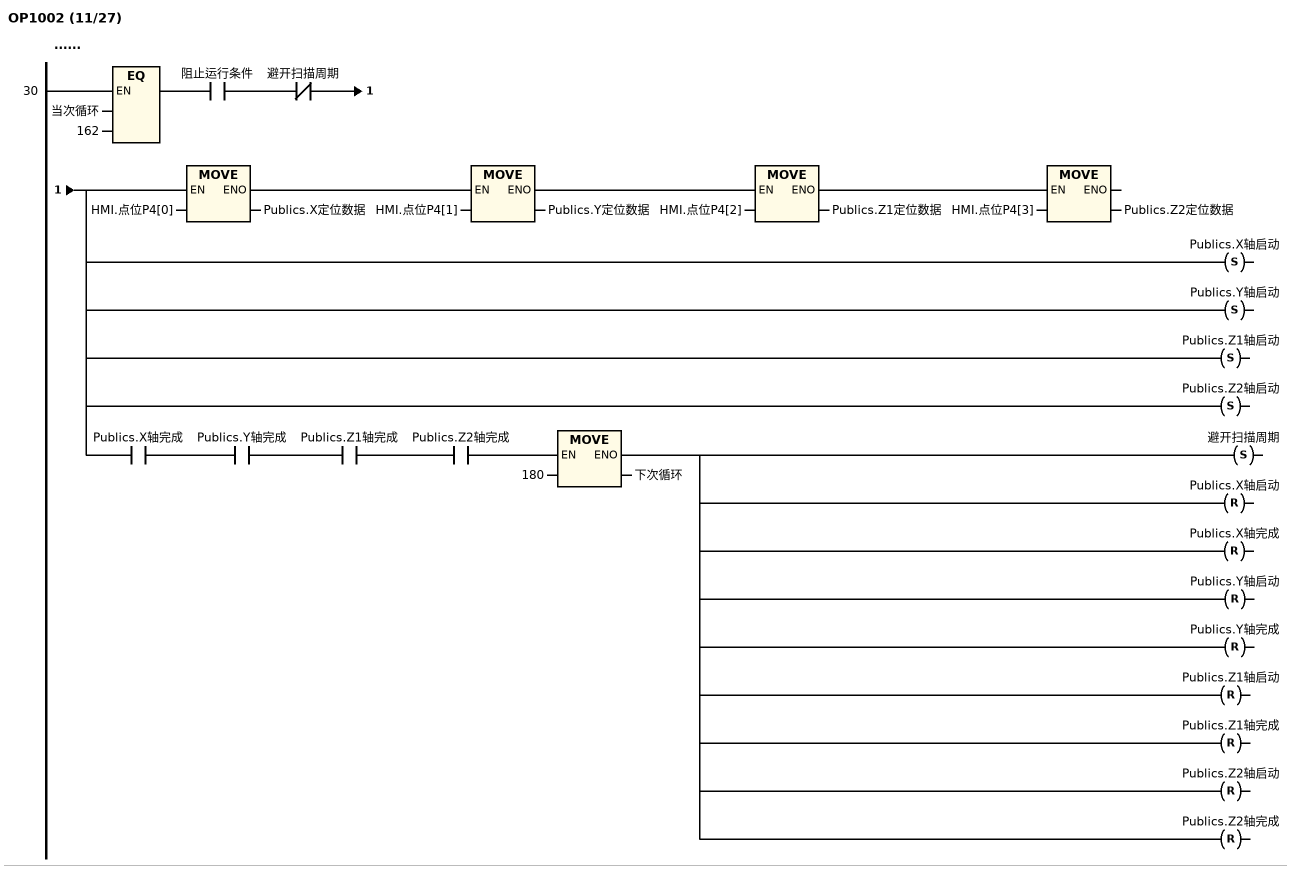
// NETWORK 30: ......
_w32 := 当次循环 = 162 AND 阻止运行条件 AND NOT 避开扫描周期;
IF _w32 THEN Publics.X定位数据 := HMI.点位P4[0]; END_IF
IF _w32 THEN Publics.Y定位数据 := HMI.点位P4[1]; END_IF
IF _w32 THEN Publics.Z1定位数据 := HMI.点位P4[2]; END_IF
IF _w32 THEN Publics.Z2定位数据 := HMI.点位P4[3]; END_IF
Publics.X轴启动 S= _w32;
Publics.Y轴启动 S= _w32;
Publics.Z1轴启动 S= _w32;
Publics.Z2轴启动 S= _w32;
IF _w32 AND Publics.X轴完成 AND Publics.Y轴完成 AND Publics.Z1轴完成 AND Publics.Z2轴完成 THEN 下次循环 := 180; END_IF
_w33 := _w32 AND Publics.X轴完成 AND Publics.Y轴完成 AND Publics.Z1轴完成 AND Publics.Z2轴完成;
避开扫描周期 S= _w33;
Publics.X轴启动 R= _w33;
Publics.X轴完成 R= _w33;
Publics.Y轴启动 R= _w33;
Publics.Y轴完成 R= _w33;
Publics.Z1轴启动 R= _w33;
Publics.Z1轴完成 R= _w33;
Publics.Z2轴启动 R= _w33;
Publics.Z2轴完成 R= _w33;

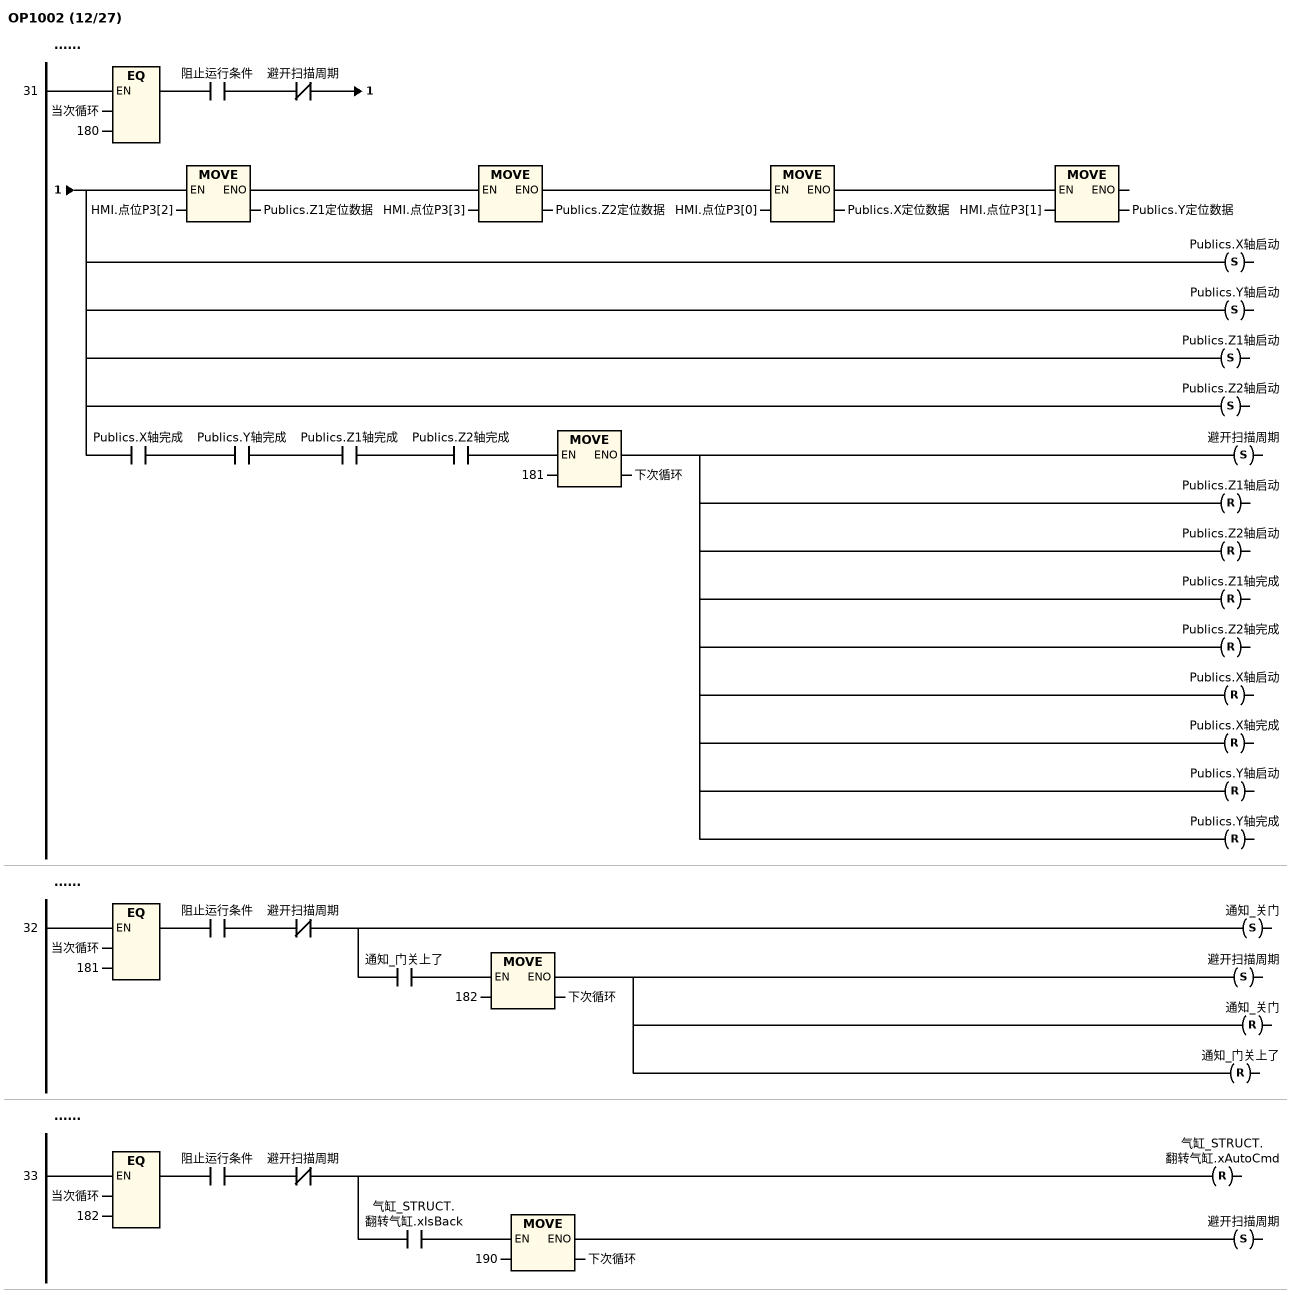
// NETWORK 31: ......
_w34 := 当次循环 = 180 AND 阻止运行条件 AND NOT 避开扫描周期;
IF _w34 THEN Publics.Z1定位数据 := HMI.点位P3[2]; END_IF
IF _w34 THEN Publics.Z2定位数据 := HMI.点位P3[3]; END_IF
IF _w34 THEN Publics.X定位数据 := HMI.点位P3[0]; END_IF
IF _w34 THEN Publics.Y定位数据 := HMI.点位P3[1]; END_IF
Publics.X轴启动 S= _w34;
Publics.Y轴启动 S= _w34;
Publics.Z1轴启动 S= _w34;
Publics.Z2轴启动 S= _w34;
IF _w34 AND Publics.X轴完成 AND Publics.Y轴完成 AND Publics.Z1轴完成 AND Publics.Z2轴完成 THEN 下次循环 := 181; END_IF
_w35 := _w34 AND Publics.X轴完成 AND Publics.Y轴完成 AND Publics.Z1轴完成 AND Publics.Z2轴完成;
避开扫描周期 S= _w35;
Publics.Z1轴启动 R= _w35;
Publics.Z2轴启动 R= _w35;
Publics.Z1轴完成 R= _w35;
Publics.Z2轴完成 R= _w35;
Publics.X轴启动 R= _w35;
Publics.X轴完成 R= _w35;
Publics.Y轴启动 R= _w35;
Publics.Y轴完成 R= _w35;

// NETWORK 32: ......
_w36 := 当次循环 = 181 AND 阻止运行条件 AND NOT 避开扫描周期;
通知_关门 S= _w36;
IF _w36 AND 通知_门关上了 THEN 下次循环 := 182; END_IF
_w37 := _w36 AND 通知_门关上了;
避开扫描周期 S= _w37;
通知_关门 R= _w37;
通知_门关上了 R= _w37;

// NETWORK 33: ......
_w38 := 当次循环 = 182 AND 阻止运行条件 AND NOT 避开扫描周期;
气缸_STRUCT.翻转气缸.xAutoCmd R= _w38;
IF _w38 AND 气缸_STRUCT.翻转气缸.xIsBack THEN 下次循环 := 190; END_IF
避开扫描周期 S= _w38 AND 气缸_STRUCT.翻转气缸.xIsBack;

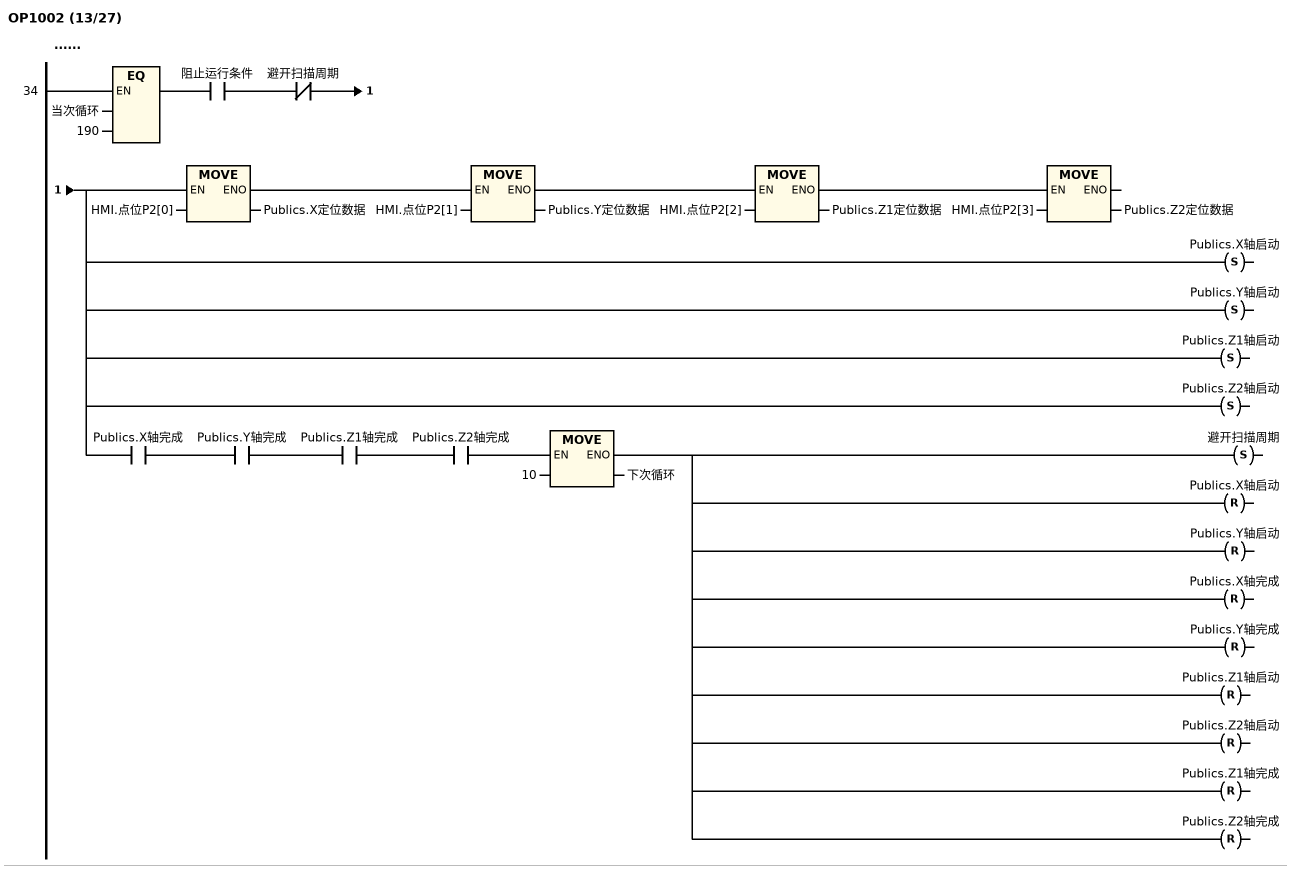
// NETWORK 34: ......
_w39 := 当次循环 = 190 AND 阻止运行条件 AND NOT 避开扫描周期;
IF _w39 THEN Publics.X定位数据 := HMI.点位P2[0]; END_IF
IF _w39 THEN Publics.Y定位数据 := HMI.点位P2[1]; END_IF
IF _w39 THEN Publics.Z1定位数据 := HMI.点位P2[2]; END_IF
IF _w39 THEN Publics.Z2定位数据 := HMI.点位P2[3]; END_IF
Publics.X轴启动 S= _w39;
Publics.Y轴启动 S= _w39;
Publics.Z1轴启动 S= _w39;
Publics.Z2轴启动 S= _w39;
IF _w39 AND Publics.X轴完成 AND Publics.Y轴完成 AND Publics.Z1轴完成 AND Publics.Z2轴完成 THEN 下次循环 := 10; END_IF
_w40 := _w39 AND Publics.X轴完成 AND Publics.Y轴完成 AND Publics.Z1轴完成 AND Publics.Z2轴完成;
避开扫描周期 S= _w40;
Publics.X轴启动 R= _w40;
Publics.Y轴启动 R= _w40;
Publics.X轴完成 R= _w40;
Publics.Y轴完成 R= _w40;
Publics.Z1轴启动 R= _w40;
Publics.Z2轴启动 R= _w40;
Publics.Z1轴完成 R= _w40;
Publics.Z2轴完成 R= _w40;

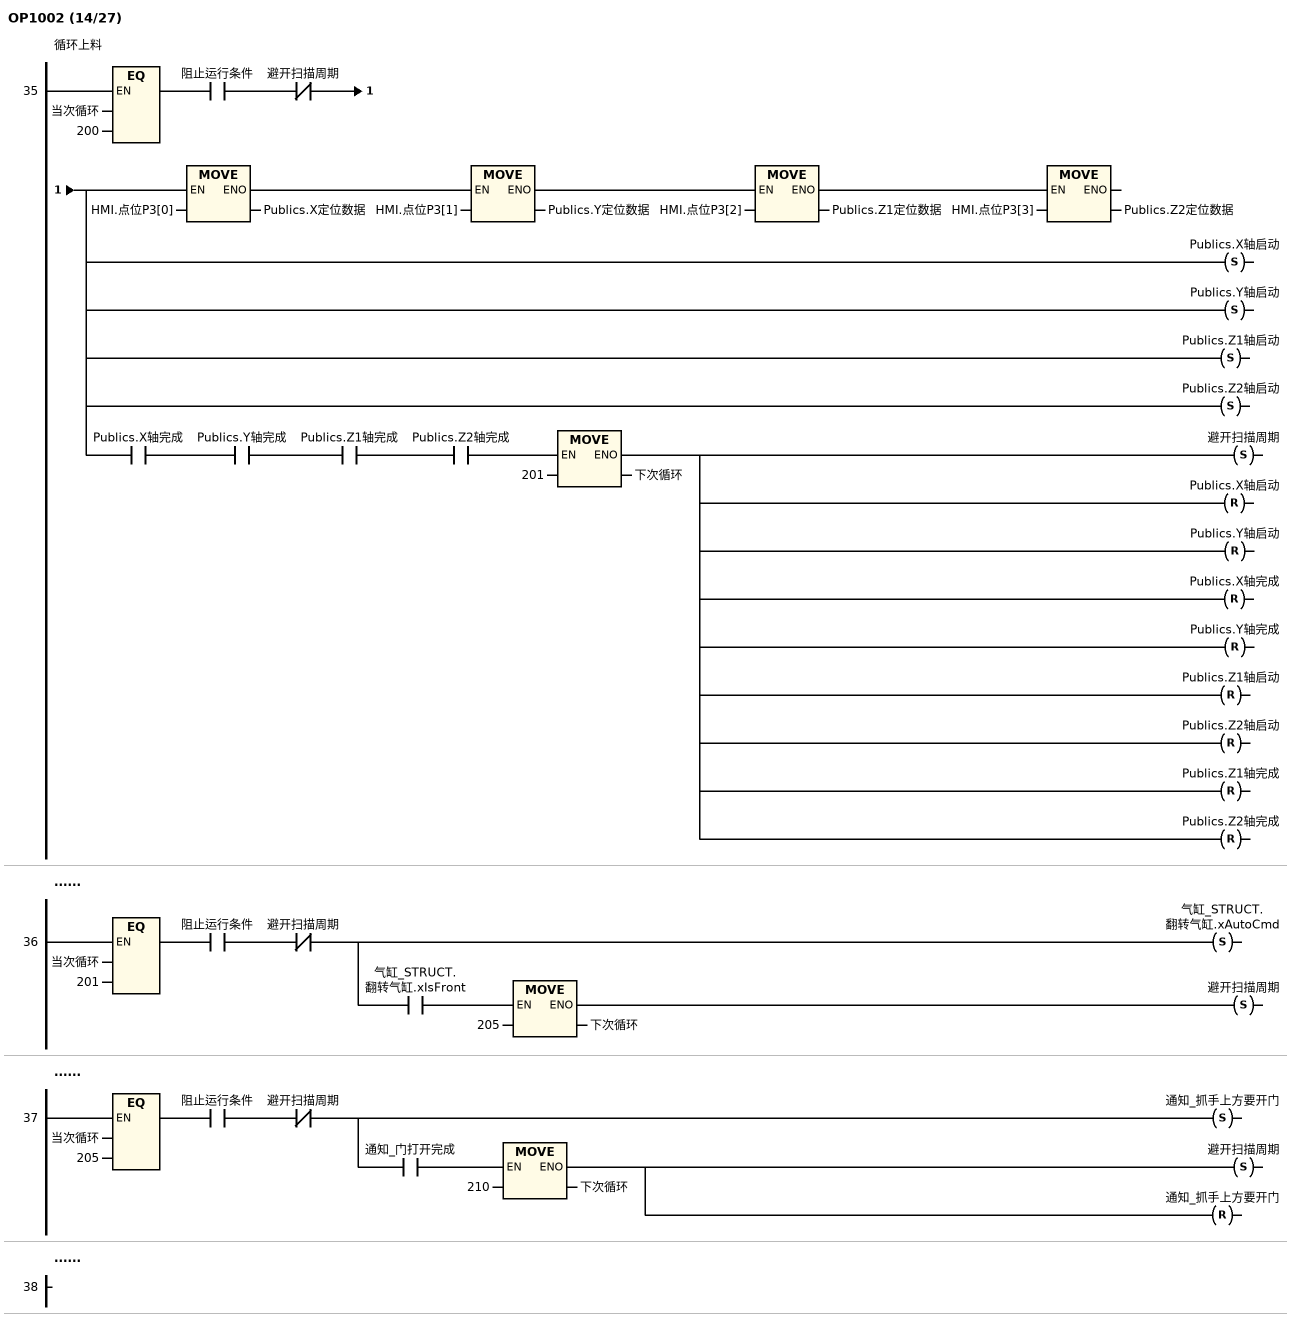
// NETWORK 35: 循环上料
_w41 := 当次循环 = 200 AND 阻止运行条件 AND NOT 避开扫描周期;
IF _w41 THEN Publics.X定位数据 := HMI.点位P3[0]; END_IF
IF _w41 THEN Publics.Y定位数据 := HMI.点位P3[1]; END_IF
IF _w41 THEN Publics.Z1定位数据 := HMI.点位P3[2]; END_IF
IF _w41 THEN Publics.Z2定位数据 := HMI.点位P3[3]; END_IF
Publics.X轴启动 S= _w41;
Publics.Y轴启动 S= _w41;
Publics.Z1轴启动 S= _w41;
Publics.Z2轴启动 S= _w41;
IF _w41 AND Publics.X轴完成 AND Publics.Y轴完成 AND Publics.Z1轴完成 AND Publics.Z2轴完成 THEN 下次循环 := 201; END_IF
_w42 := _w41 AND Publics.X轴完成 AND Publics.Y轴完成 AND Publics.Z1轴完成 AND Publics.Z2轴完成;
避开扫描周期 S= _w42;
Publics.X轴启动 R= _w42;
Publics.Y轴启动 R= _w42;
Publics.X轴完成 R= _w42;
Publics.Y轴完成 R= _w42;
Publics.Z1轴启动 R= _w42;
Publics.Z2轴启动 R= _w42;
Publics.Z1轴完成 R= _w42;
Publics.Z2轴完成 R= _w42;

// NETWORK 36: ......
_w43 := 当次循环 = 201 AND 阻止运行条件 AND NOT 避开扫描周期;
气缸_STRUCT.翻转气缸.xAutoCmd S= _w43;
IF _w43 AND 气缸_STRUCT.翻转气缸.xIsFront THEN 下次循环 := 205; END_IF
避开扫描周期 S= _w43 AND 气缸_STRUCT.翻转气缸.xIsFront;

// NETWORK 37: ......
_w44 := 当次循环 = 205 AND 阻止运行条件 AND NOT 避开扫描周期;
通知_抓手上方要开门 S= _w44;
IF _w44 AND 通知_门打开完成 THEN 下次循环 := 210; END_IF
_w45 := _w44 AND 通知_门打开完成;
避开扫描周期 S= _w45;
通知_抓手上方要开门 R= _w45;

// NETWORK 38: ......

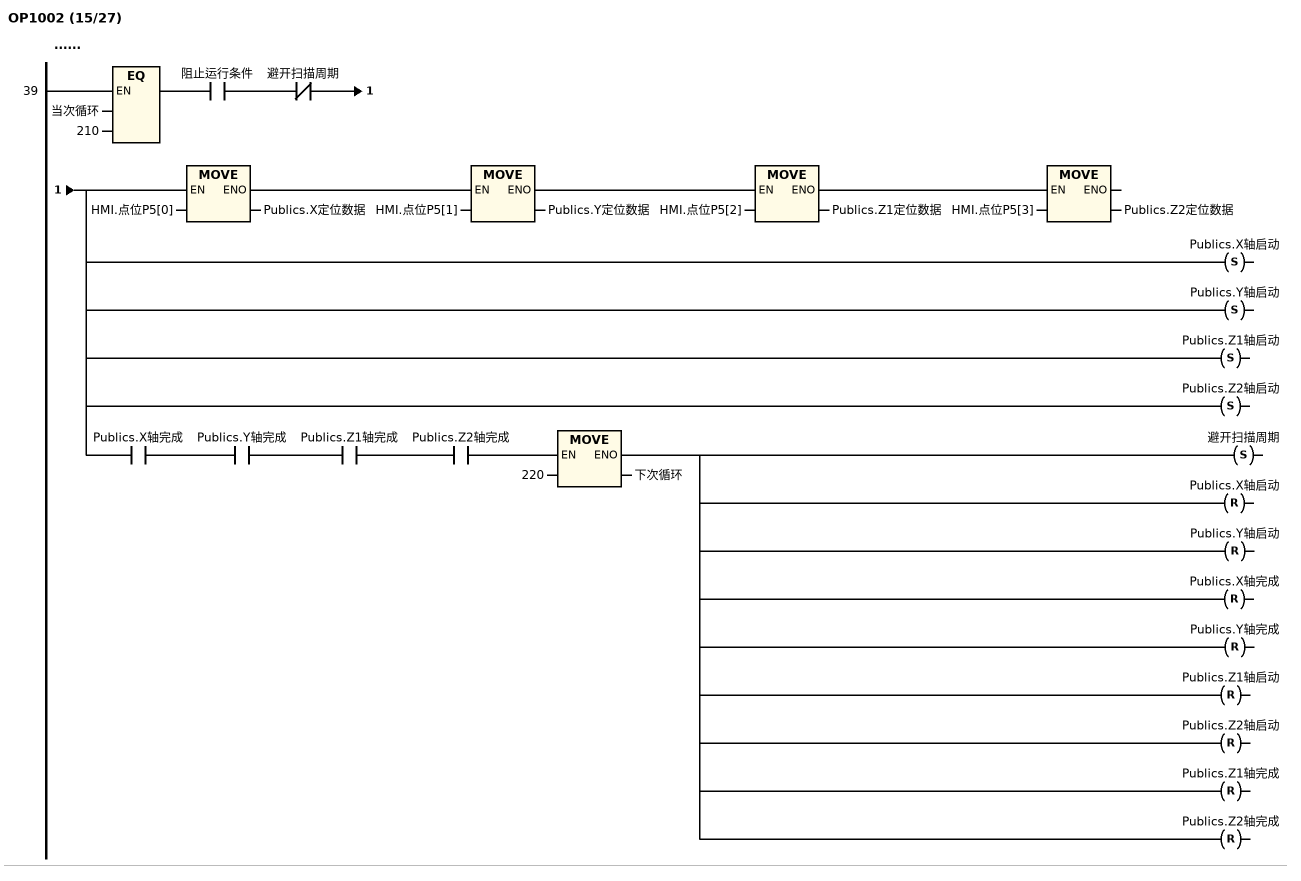
// NETWORK 39: ......
_w46 := 当次循环 = 210 AND 阻止运行条件 AND NOT 避开扫描周期;
IF _w46 THEN Publics.X定位数据 := HMI.点位P5[0]; END_IF
IF _w46 THEN Publics.Y定位数据 := HMI.点位P5[1]; END_IF
IF _w46 THEN Publics.Z1定位数据 := HMI.点位P5[2]; END_IF
IF _w46 THEN Publics.Z2定位数据 := HMI.点位P5[3]; END_IF
Publics.X轴启动 S= _w46;
Publics.Y轴启动 S= _w46;
Publics.Z1轴启动 S= _w46;
Publics.Z2轴启动 S= _w46;
IF _w46 AND Publics.X轴完成 AND Publics.Y轴完成 AND Publics.Z1轴完成 AND Publics.Z2轴完成 THEN 下次循环 := 220; END_IF
_w47 := _w46 AND Publics.X轴完成 AND Publics.Y轴完成 AND Publics.Z1轴完成 AND Publics.Z2轴完成;
避开扫描周期 S= _w47;
Publics.X轴启动 R= _w47;
Publics.Y轴启动 R= _w47;
Publics.X轴完成 R= _w47;
Publics.Y轴完成 R= _w47;
Publics.Z1轴启动 R= _w47;
Publics.Z2轴启动 R= _w47;
Publics.Z1轴完成 R= _w47;
Publics.Z2轴完成 R= _w47;

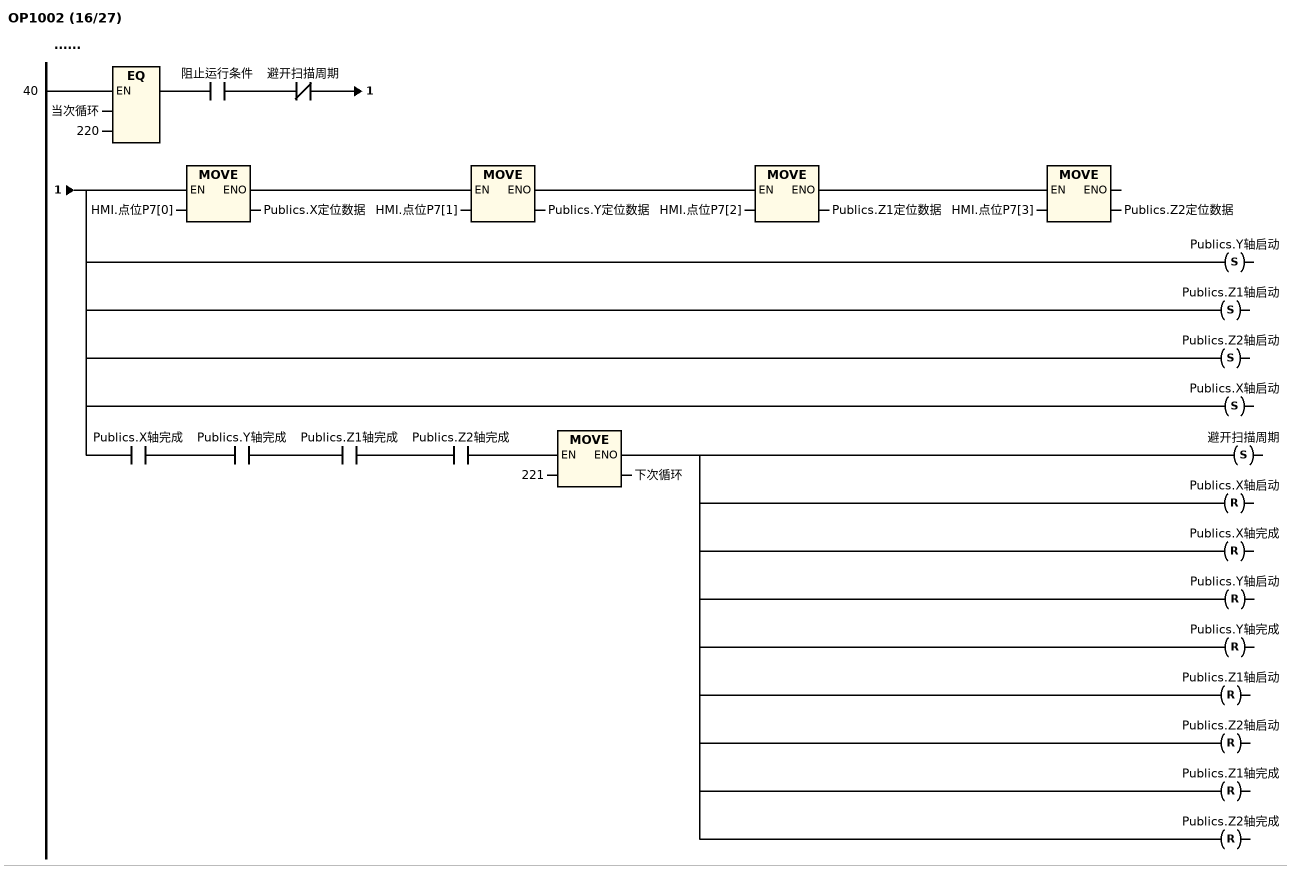
// NETWORK 40: ......
_w48 := 当次循环 = 220 AND 阻止运行条件 AND NOT 避开扫描周期;
IF _w48 THEN Publics.X定位数据 := HMI.点位P7[0]; END_IF
IF _w48 THEN Publics.Y定位数据 := HMI.点位P7[1]; END_IF
IF _w48 THEN Publics.Z1定位数据 := HMI.点位P7[2]; END_IF
IF _w48 THEN Publics.Z2定位数据 := HMI.点位P7[3]; END_IF
Publics.Y轴启动 S= _w48;
Publics.Z1轴启动 S= _w48;
Publics.Z2轴启动 S= _w48;
Publics.X轴启动 S= _w48;
IF _w48 AND Publics.X轴完成 AND Publics.Y轴完成 AND Publics.Z1轴完成 AND Publics.Z2轴完成 THEN 下次循环 := 221; END_IF
_w49 := _w48 AND Publics.X轴完成 AND Publics.Y轴完成 AND Publics.Z1轴完成 AND Publics.Z2轴完成;
避开扫描周期 S= _w49;
Publics.X轴启动 R= _w49;
Publics.X轴完成 R= _w49;
Publics.Y轴启动 R= _w49;
Publics.Y轴完成 R= _w49;
Publics.Z1轴启动 R= _w49;
Publics.Z2轴启动 R= _w49;
Publics.Z1轴完成 R= _w49;
Publics.Z2轴完成 R= _w49;

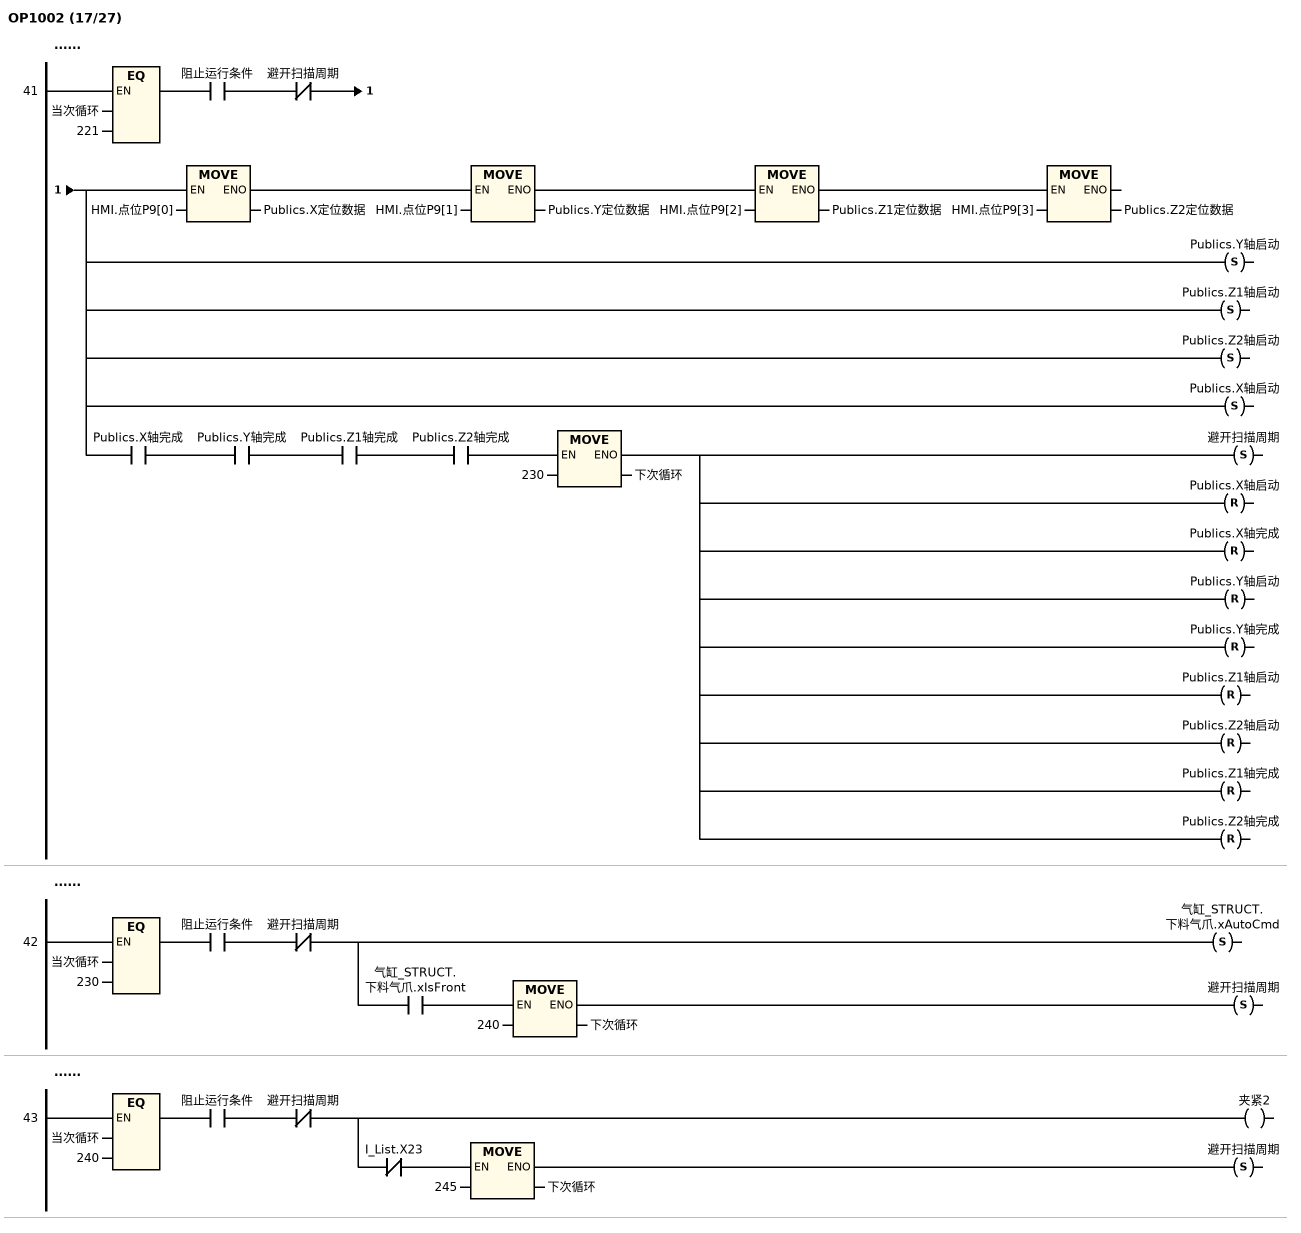
// NETWORK 41: ......
_w50 := 当次循环 = 221 AND 阻止运行条件 AND NOT 避开扫描周期;
IF _w50 THEN Publics.X定位数据 := HMI.点位P9[0]; END_IF
IF _w50 THEN Publics.Y定位数据 := HMI.点位P9[1]; END_IF
IF _w50 THEN Publics.Z1定位数据 := HMI.点位P9[2]; END_IF
IF _w50 THEN Publics.Z2定位数据 := HMI.点位P9[3]; END_IF
Publics.Y轴启动 S= _w50;
Publics.Z1轴启动 S= _w50;
Publics.Z2轴启动 S= _w50;
Publics.X轴启动 S= _w50;
IF _w50 AND Publics.X轴完成 AND Publics.Y轴完成 AND Publics.Z1轴完成 AND Publics.Z2轴完成 THEN 下次循环 := 230; END_IF
_w51 := _w50 AND Publics.X轴完成 AND Publics.Y轴完成 AND Publics.Z1轴完成 AND Publics.Z2轴完成;
避开扫描周期 S= _w51;
Publics.X轴启动 R= _w51;
Publics.X轴完成 R= _w51;
Publics.Y轴启动 R= _w51;
Publics.Y轴完成 R= _w51;
Publics.Z1轴启动 R= _w51;
Publics.Z2轴启动 R= _w51;
Publics.Z1轴完成 R= _w51;
Publics.Z2轴完成 R= _w51;

// NETWORK 42: ......
_w52 := 当次循环 = 230 AND 阻止运行条件 AND NOT 避开扫描周期;
气缸_STRUCT.下料气爪.xAutoCmd S= _w52;
IF _w52 AND 气缸_STRUCT.下料气爪.xIsFront THEN 下次循环 := 240; END_IF
避开扫描周期 S= _w52 AND 气缸_STRUCT.下料气爪.xIsFront;

// NETWORK 43: ......
_w53 := 当次循环 = 240 AND 阻止运行条件 AND NOT 避开扫描周期;
夹紧2 := _w53;
IF _w53 AND NOT I_List.X23 THEN 下次循环 := 245; END_IF
避开扫描周期 S= _w53 AND NOT I_List.X23;

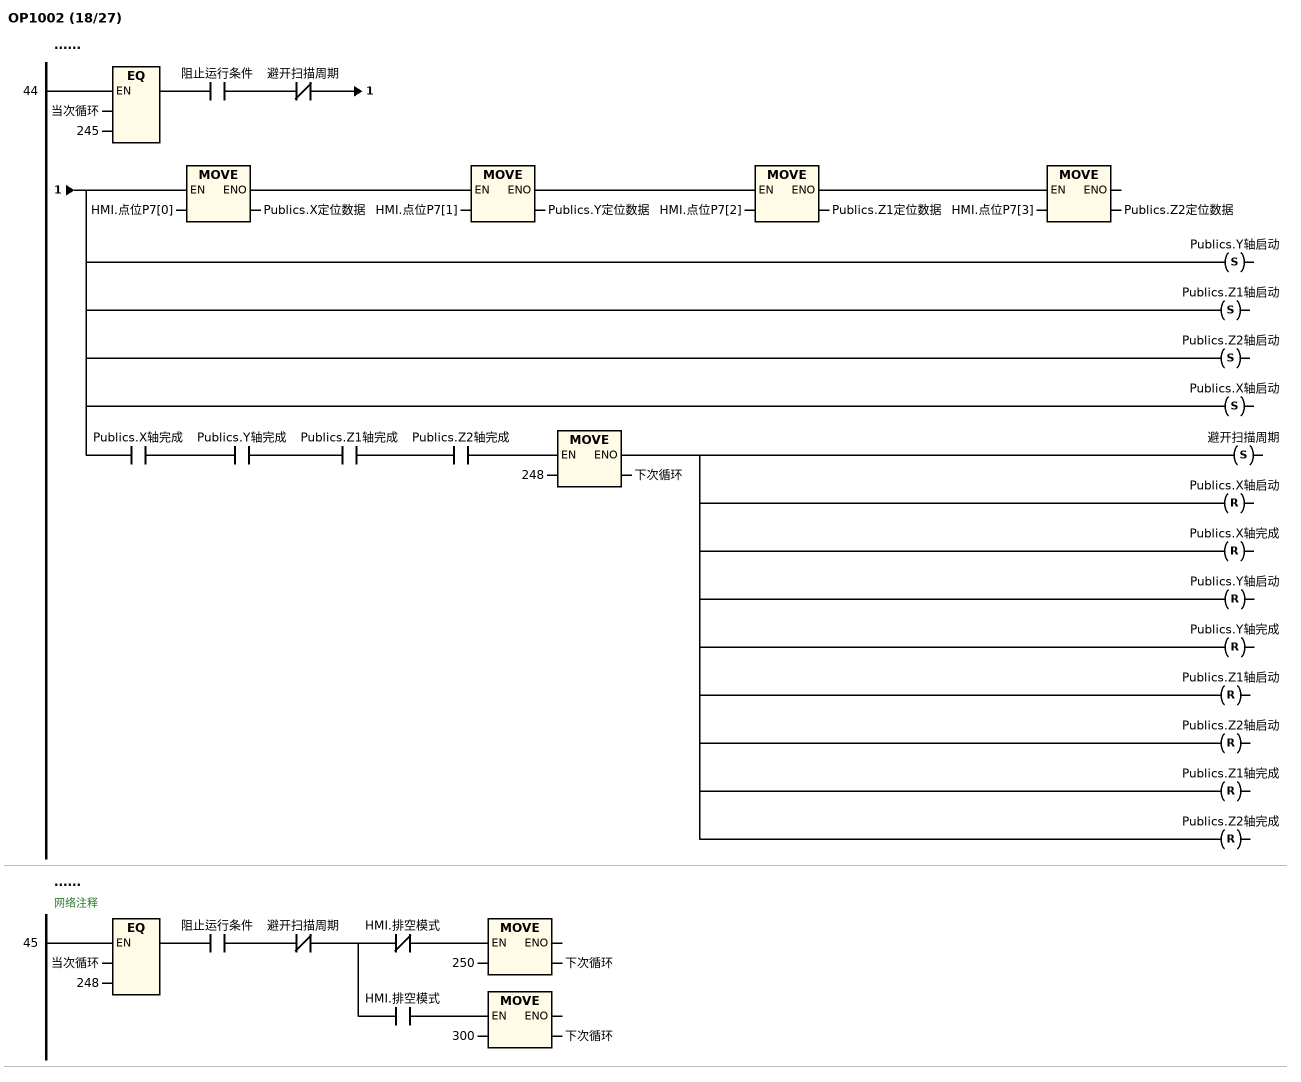
// NETWORK 44: ......
_w54 := 当次循环 = 245 AND 阻止运行条件 AND NOT 避开扫描周期;
IF _w54 THEN Publics.X定位数据 := HMI.点位P7[0]; END_IF
IF _w54 THEN Publics.Y定位数据 := HMI.点位P7[1]; END_IF
IF _w54 THEN Publics.Z1定位数据 := HMI.点位P7[2]; END_IF
IF _w54 THEN Publics.Z2定位数据 := HMI.点位P7[3]; END_IF
Publics.Y轴启动 S= _w54;
Publics.Z1轴启动 S= _w54;
Publics.Z2轴启动 S= _w54;
Publics.X轴启动 S= _w54;
IF _w54 AND Publics.X轴完成 AND Publics.Y轴完成 AND Publics.Z1轴完成 AND Publics.Z2轴完成 THEN 下次循环 := 248; END_IF
_w55 := _w54 AND Publics.X轴完成 AND Publics.Y轴完成 AND Publics.Z1轴完成 AND Publics.Z2轴完成;
避开扫描周期 S= _w55;
Publics.X轴启动 R= _w55;
Publics.X轴完成 R= _w55;
Publics.Y轴启动 R= _w55;
Publics.Y轴完成 R= _w55;
Publics.Z1轴启动 R= _w55;
Publics.Z2轴启动 R= _w55;
Publics.Z1轴完成 R= _w55;
Publics.Z2轴完成 R= _w55;

// NETWORK 45: ......
// 网络注释
_w56 := 当次循环 = 248 AND 阻止运行条件 AND NOT 避开扫描周期;
IF _w56 AND NOT HMI.排空模式 THEN 下次循环 := 250; END_IF
IF _w56 AND HMI.排空模式 THEN 下次循环 := 300; END_IF

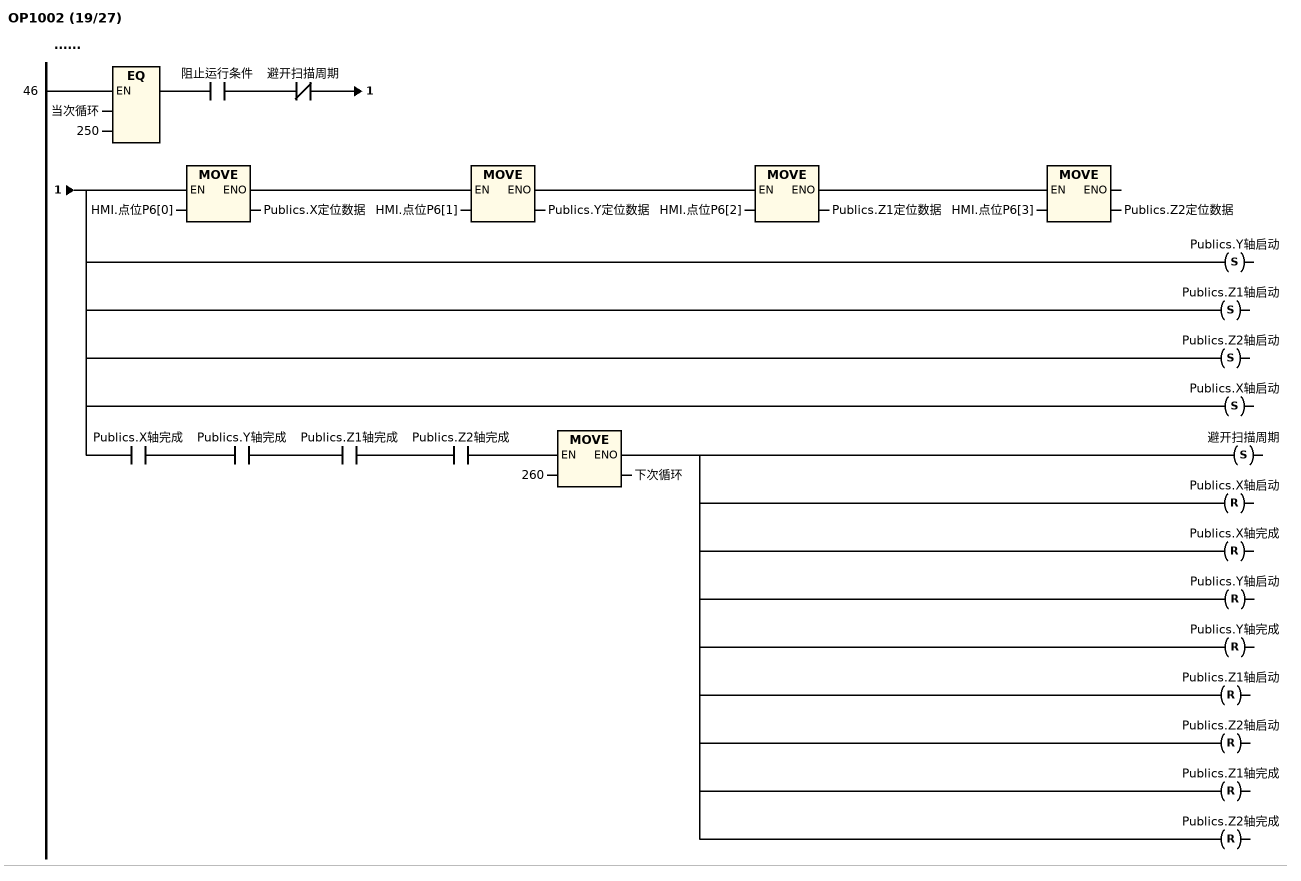
// NETWORK 46: ......
_w57 := 当次循环 = 250 AND 阻止运行条件 AND NOT 避开扫描周期;
IF _w57 THEN Publics.X定位数据 := HMI.点位P6[0]; END_IF
IF _w57 THEN Publics.Y定位数据 := HMI.点位P6[1]; END_IF
IF _w57 THEN Publics.Z1定位数据 := HMI.点位P6[2]; END_IF
IF _w57 THEN Publics.Z2定位数据 := HMI.点位P6[3]; END_IF
Publics.Y轴启动 S= _w57;
Publics.Z1轴启动 S= _w57;
Publics.Z2轴启动 S= _w57;
Publics.X轴启动 S= _w57;
IF _w57 AND Publics.X轴完成 AND Publics.Y轴完成 AND Publics.Z1轴完成 AND Publics.Z2轴完成 THEN 下次循环 := 260; END_IF
_w58 := _w57 AND Publics.X轴完成 AND Publics.Y轴完成 AND Publics.Z1轴完成 AND Publics.Z2轴完成;
避开扫描周期 S= _w58;
Publics.X轴启动 R= _w58;
Publics.X轴完成 R= _w58;
Publics.Y轴启动 R= _w58;
Publics.Y轴完成 R= _w58;
Publics.Z1轴启动 R= _w58;
Publics.Z2轴启动 R= _w58;
Publics.Z1轴完成 R= _w58;
Publics.Z2轴完成 R= _w58;

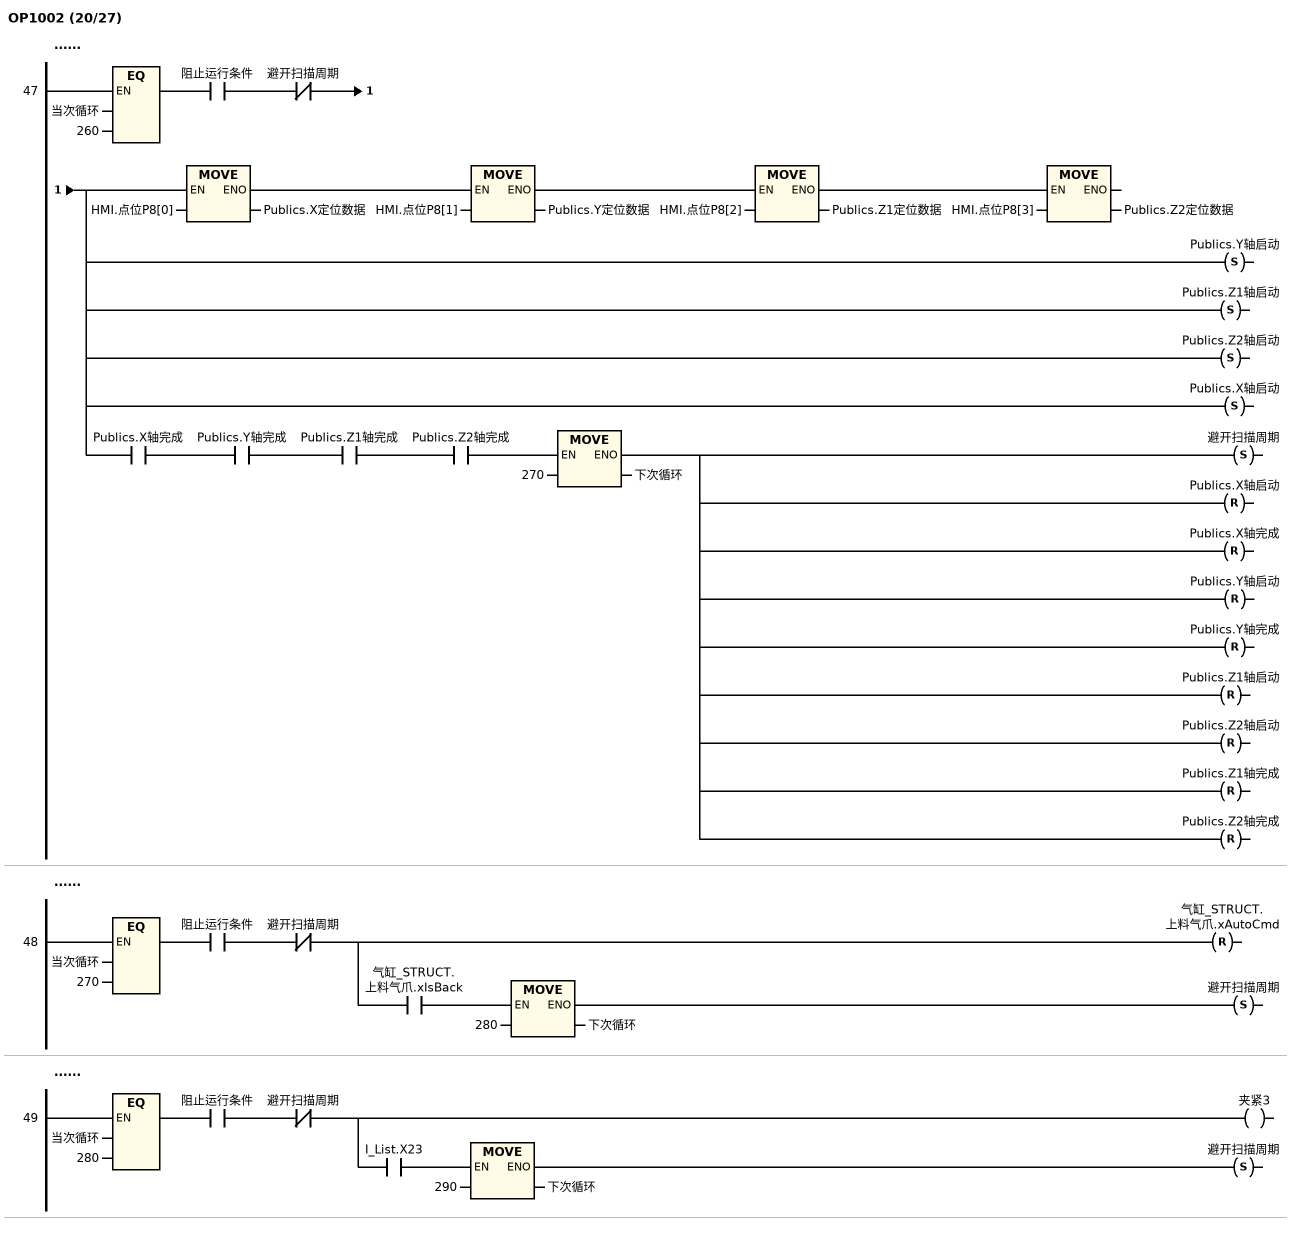
// NETWORK 47: ......
_w59 := 当次循环 = 260 AND 阻止运行条件 AND NOT 避开扫描周期;
IF _w59 THEN Publics.X定位数据 := HMI.点位P8[0]; END_IF
IF _w59 THEN Publics.Y定位数据 := HMI.点位P8[1]; END_IF
IF _w59 THEN Publics.Z1定位数据 := HMI.点位P8[2]; END_IF
IF _w59 THEN Publics.Z2定位数据 := HMI.点位P8[3]; END_IF
Publics.Y轴启动 S= _w59;
Publics.Z1轴启动 S= _w59;
Publics.Z2轴启动 S= _w59;
Publics.X轴启动 S= _w59;
IF _w59 AND Publics.X轴完成 AND Publics.Y轴完成 AND Publics.Z1轴完成 AND Publics.Z2轴完成 THEN 下次循环 := 270; END_IF
_w60 := _w59 AND Publics.X轴完成 AND Publics.Y轴完成 AND Publics.Z1轴完成 AND Publics.Z2轴完成;
避开扫描周期 S= _w60;
Publics.X轴启动 R= _w60;
Publics.X轴完成 R= _w60;
Publics.Y轴启动 R= _w60;
Publics.Y轴完成 R= _w60;
Publics.Z1轴启动 R= _w60;
Publics.Z2轴启动 R= _w60;
Publics.Z1轴完成 R= _w60;
Publics.Z2轴完成 R= _w60;

// NETWORK 48: ......
_w61 := 当次循环 = 270 AND 阻止运行条件 AND NOT 避开扫描周期;
气缸_STRUCT.上料气爪.xAutoCmd R= _w61;
IF _w61 AND 气缸_STRUCT.上料气爪.xIsBack THEN 下次循环 := 280; END_IF
避开扫描周期 S= _w61 AND 气缸_STRUCT.上料气爪.xIsBack;

// NETWORK 49: ......
_w62 := 当次循环 = 280 AND 阻止运行条件 AND NOT 避开扫描周期;
夹紧3 := _w62;
IF _w62 AND I_List.X23 THEN 下次循环 := 290; END_IF
避开扫描周期 S= _w62 AND I_List.X23;

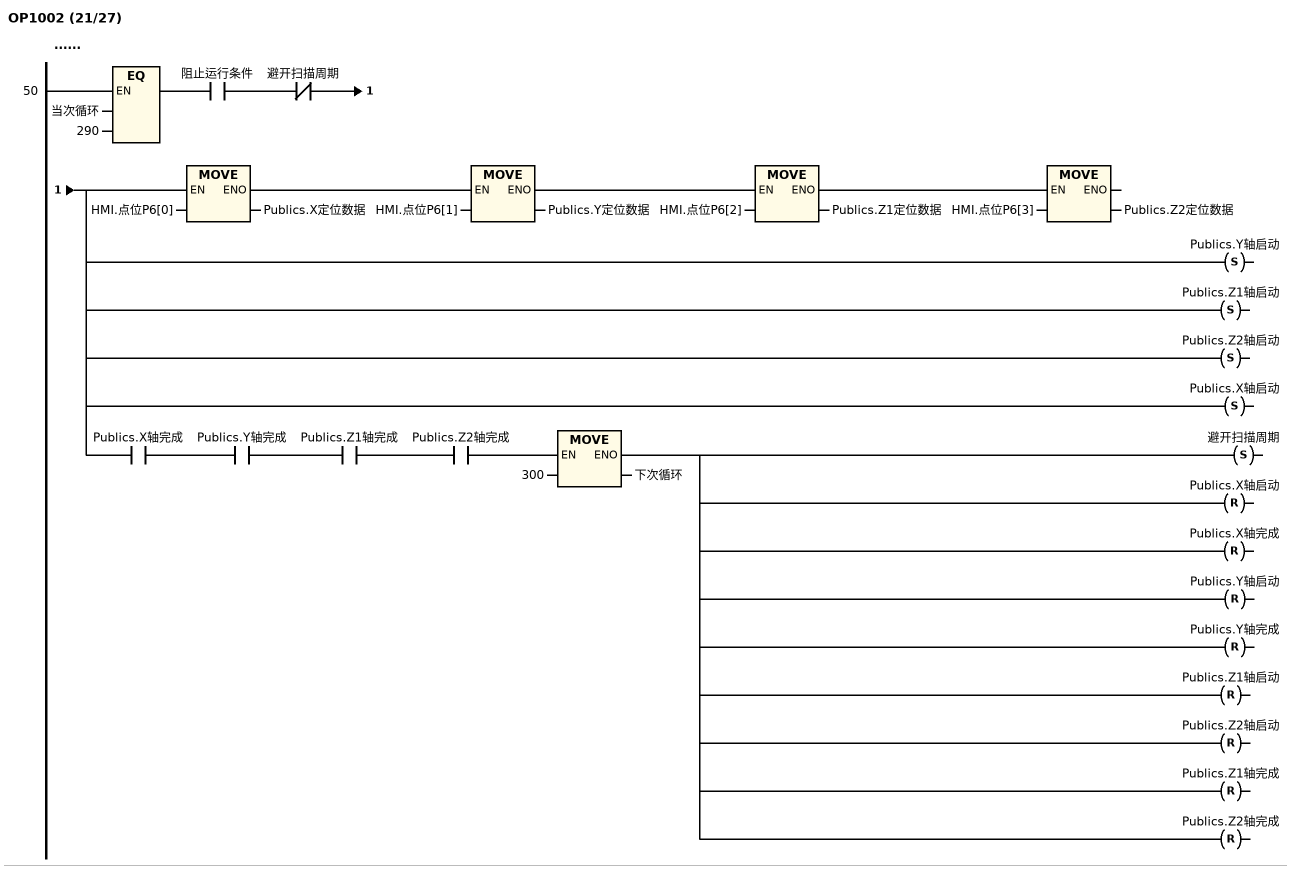
// NETWORK 50: ......
_w63 := 当次循环 = 290 AND 阻止运行条件 AND NOT 避开扫描周期;
IF _w63 THEN Publics.X定位数据 := HMI.点位P6[0]; END_IF
IF _w63 THEN Publics.Y定位数据 := HMI.点位P6[1]; END_IF
IF _w63 THEN Publics.Z1定位数据 := HMI.点位P6[2]; END_IF
IF _w63 THEN Publics.Z2定位数据 := HMI.点位P6[3]; END_IF
Publics.Y轴启动 S= _w63;
Publics.Z1轴启动 S= _w63;
Publics.Z2轴启动 S= _w63;
Publics.X轴启动 S= _w63;
IF _w63 AND Publics.X轴完成 AND Publics.Y轴完成 AND Publics.Z1轴完成 AND Publics.Z2轴完成 THEN 下次循环 := 300; END_IF
_w64 := _w63 AND Publics.X轴完成 AND Publics.Y轴完成 AND Publics.Z1轴完成 AND Publics.Z2轴完成;
避开扫描周期 S= _w64;
Publics.X轴启动 R= _w64;
Publics.X轴完成 R= _w64;
Publics.Y轴启动 R= _w64;
Publics.Y轴完成 R= _w64;
Publics.Z1轴启动 R= _w64;
Publics.Z2轴启动 R= _w64;
Publics.Z1轴完成 R= _w64;
Publics.Z2轴完成 R= _w64;

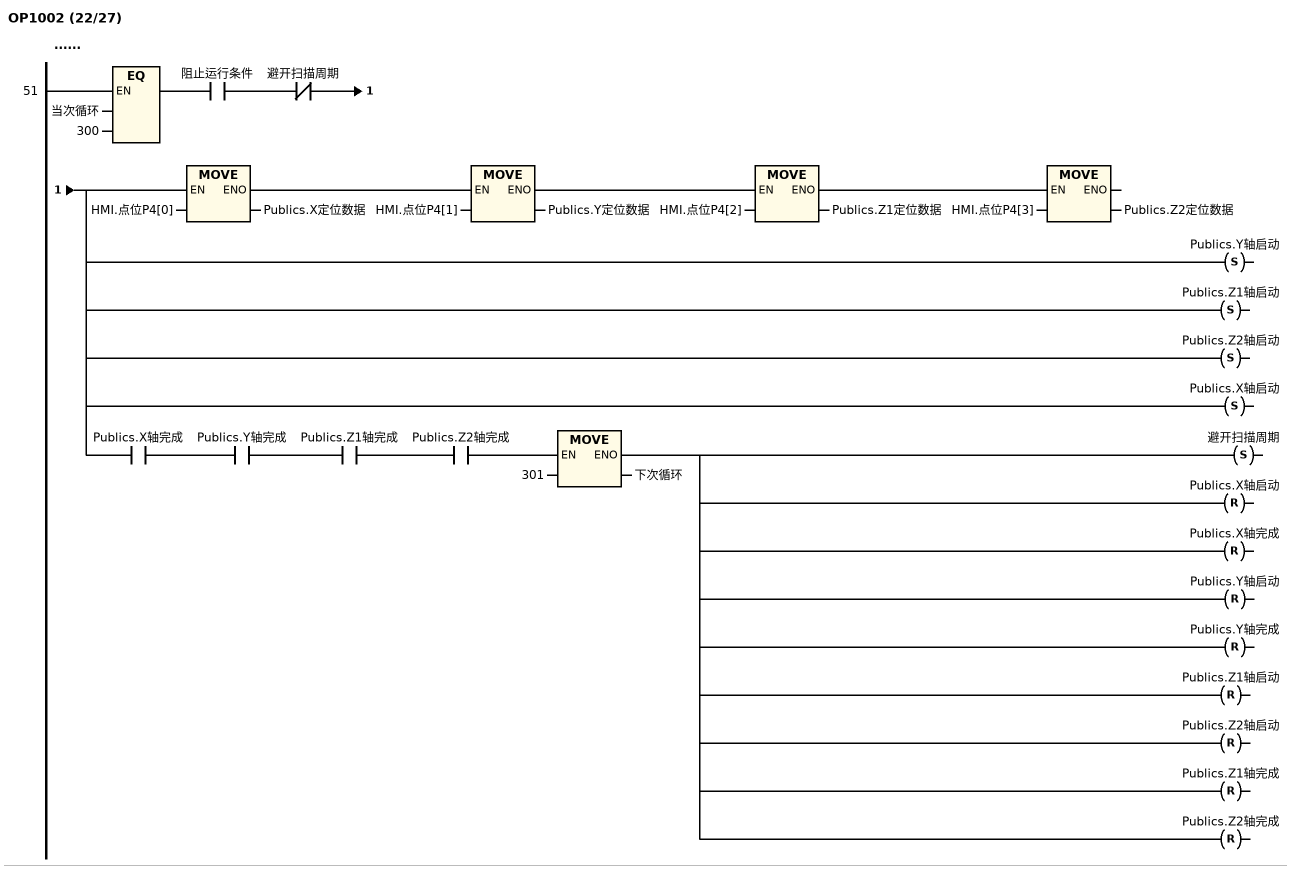
// NETWORK 51: ......
_w65 := 当次循环 = 300 AND 阻止运行条件 AND NOT 避开扫描周期;
IF _w65 THEN Publics.X定位数据 := HMI.点位P4[0]; END_IF
IF _w65 THEN Publics.Y定位数据 := HMI.点位P4[1]; END_IF
IF _w65 THEN Publics.Z1定位数据 := HMI.点位P4[2]; END_IF
IF _w65 THEN Publics.Z2定位数据 := HMI.点位P4[3]; END_IF
Publics.Y轴启动 S= _w65;
Publics.Z1轴启动 S= _w65;
Publics.Z2轴启动 S= _w65;
Publics.X轴启动 S= _w65;
IF _w65 AND Publics.X轴完成 AND Publics.Y轴完成 AND Publics.Z1轴完成 AND Publics.Z2轴完成 THEN 下次循环 := 301; END_IF
_w66 := _w65 AND Publics.X轴完成 AND Publics.Y轴完成 AND Publics.Z1轴完成 AND Publics.Z2轴完成;
避开扫描周期 S= _w66;
Publics.X轴启动 R= _w66;
Publics.X轴完成 R= _w66;
Publics.Y轴启动 R= _w66;
Publics.Y轴完成 R= _w66;
Publics.Z1轴启动 R= _w66;
Publics.Z2轴启动 R= _w66;
Publics.Z1轴完成 R= _w66;
Publics.Z2轴完成 R= _w66;

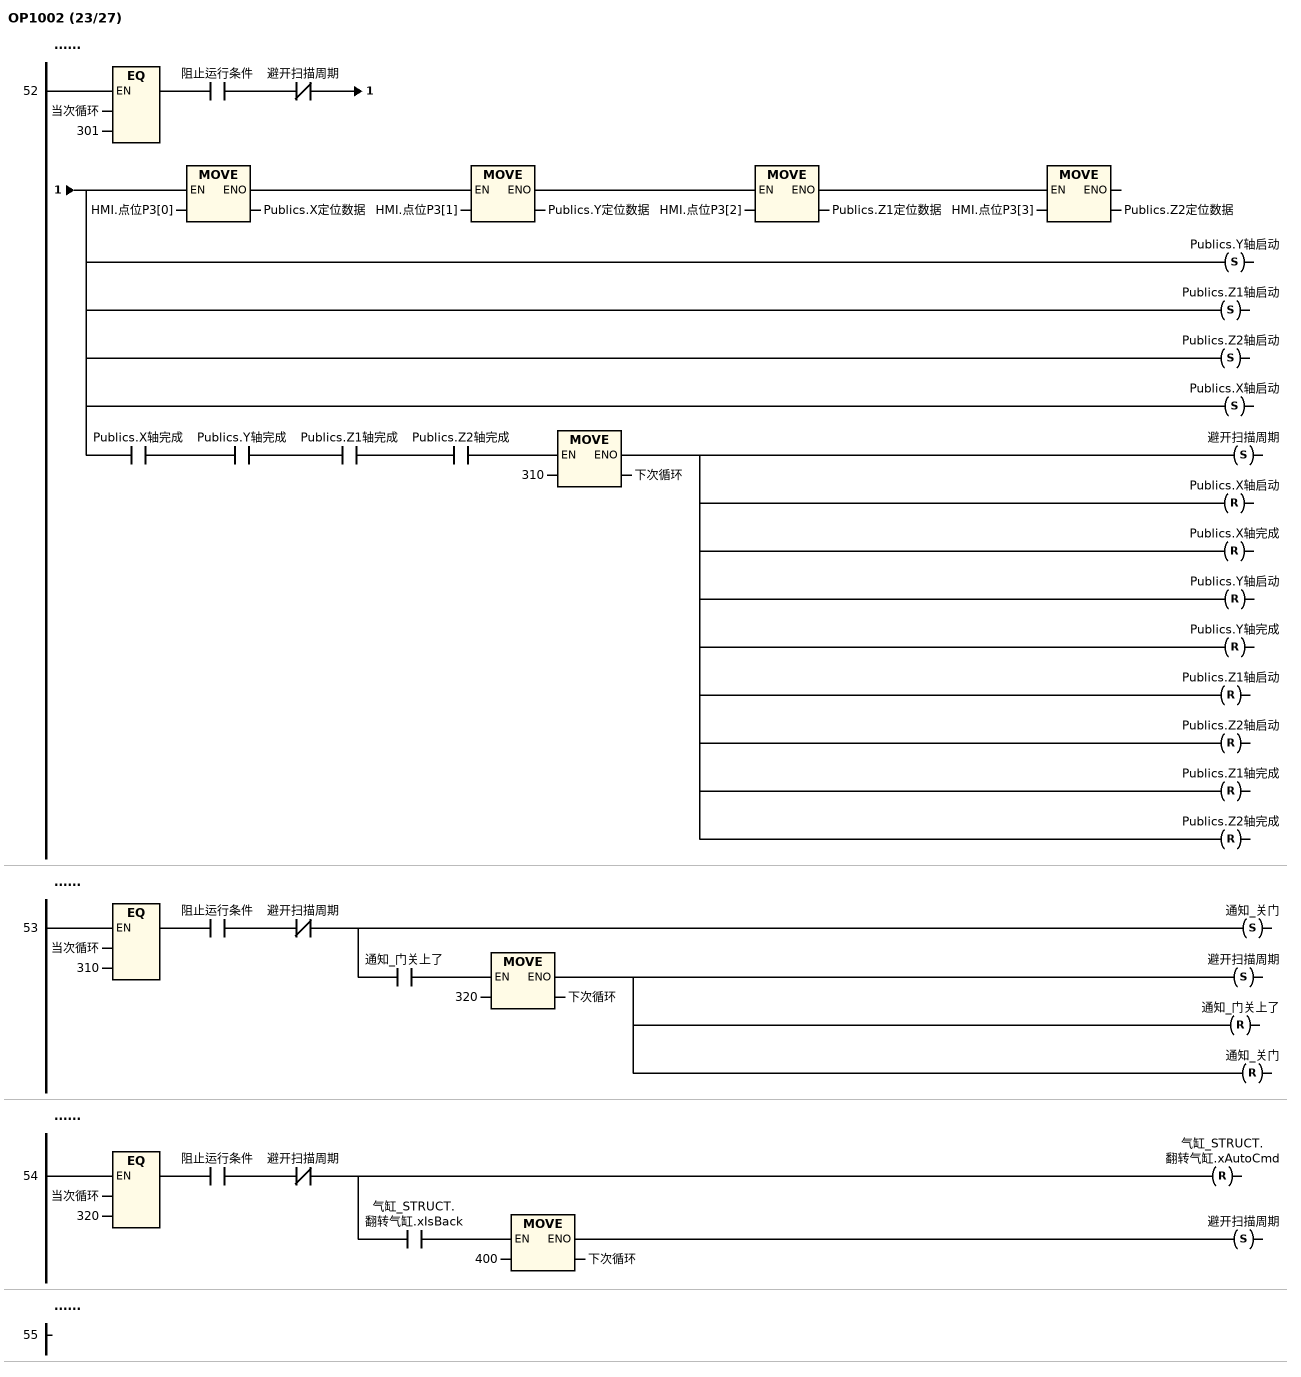
// NETWORK 52: ......
_w67 := 当次循环 = 301 AND 阻止运行条件 AND NOT 避开扫描周期;
IF _w67 THEN Publics.X定位数据 := HMI.点位P3[0]; END_IF
IF _w67 THEN Publics.Y定位数据 := HMI.点位P3[1]; END_IF
IF _w67 THEN Publics.Z1定位数据 := HMI.点位P3[2]; END_IF
IF _w67 THEN Publics.Z2定位数据 := HMI.点位P3[3]; END_IF
Publics.Y轴启动 S= _w67;
Publics.Z1轴启动 S= _w67;
Publics.Z2轴启动 S= _w67;
Publics.X轴启动 S= _w67;
IF _w67 AND Publics.X轴完成 AND Publics.Y轴完成 AND Publics.Z1轴完成 AND Publics.Z2轴完成 THEN 下次循环 := 310; END_IF
_w68 := _w67 AND Publics.X轴完成 AND Publics.Y轴完成 AND Publics.Z1轴完成 AND Publics.Z2轴完成;
避开扫描周期 S= _w68;
Publics.X轴启动 R= _w68;
Publics.X轴完成 R= _w68;
Publics.Y轴启动 R= _w68;
Publics.Y轴完成 R= _w68;
Publics.Z1轴启动 R= _w68;
Publics.Z2轴启动 R= _w68;
Publics.Z1轴完成 R= _w68;
Publics.Z2轴完成 R= _w68;

// NETWORK 53: ......
_w69 := 当次循环 = 310 AND 阻止运行条件 AND NOT 避开扫描周期;
通知_关门 S= _w69;
IF _w69 AND 通知_门关上了 THEN 下次循环 := 320; END_IF
_w70 := _w69 AND 通知_门关上了;
避开扫描周期 S= _w70;
通知_门关上了 R= _w70;
通知_关门 R= _w70;

// NETWORK 54: ......
_w71 := 当次循环 = 320 AND 阻止运行条件 AND NOT 避开扫描周期;
气缸_STRUCT.翻转气缸.xAutoCmd R= _w71;
IF _w71 AND 气缸_STRUCT.翻转气缸.xIsBack THEN 下次循环 := 400; END_IF
避开扫描周期 S= _w71 AND 气缸_STRUCT.翻转气缸.xIsBack;

// NETWORK 55: ......

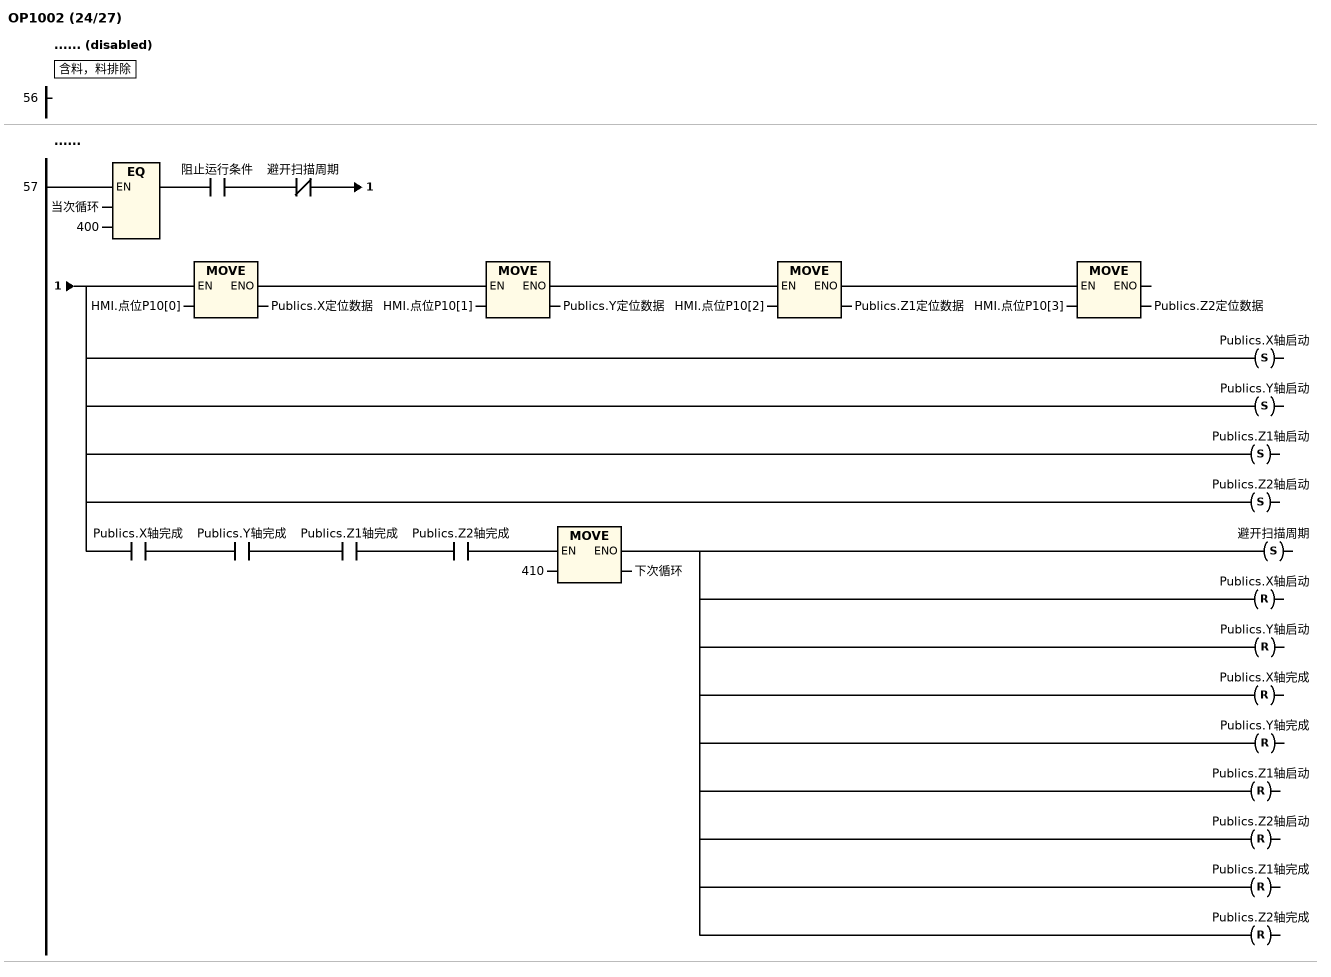
// NETWORK 56: ...... (disabled)
// label: 含料，料排除

// NETWORK 57: ......
_w72 := 当次循环 = 400 AND 阻止运行条件 AND NOT 避开扫描周期;
IF _w72 THEN Publics.X定位数据 := HMI.点位P10[0]; END_IF
IF _w72 THEN Publics.Y定位数据 := HMI.点位P10[1]; END_IF
IF _w72 THEN Publics.Z1定位数据 := HMI.点位P10[2]; END_IF
IF _w72 THEN Publics.Z2定位数据 := HMI.点位P10[3]; END_IF
Publics.X轴启动 S= _w72;
Publics.Y轴启动 S= _w72;
Publics.Z1轴启动 S= _w72;
Publics.Z2轴启动 S= _w72;
IF _w72 AND Publics.X轴完成 AND Publics.Y轴完成 AND Publics.Z1轴完成 AND Publics.Z2轴完成 THEN 下次循环 := 410; END_IF
_w73 := _w72 AND Publics.X轴完成 AND Publics.Y轴完成 AND Publics.Z1轴完成 AND Publics.Z2轴完成;
避开扫描周期 S= _w73;
Publics.X轴启动 R= _w73;
Publics.Y轴启动 R= _w73;
Publics.X轴完成 R= _w73;
Publics.Y轴完成 R= _w73;
Publics.Z1轴启动 R= _w73;
Publics.Z2轴启动 R= _w73;
Publics.Z1轴完成 R= _w73;
Publics.Z2轴完成 R= _w73;

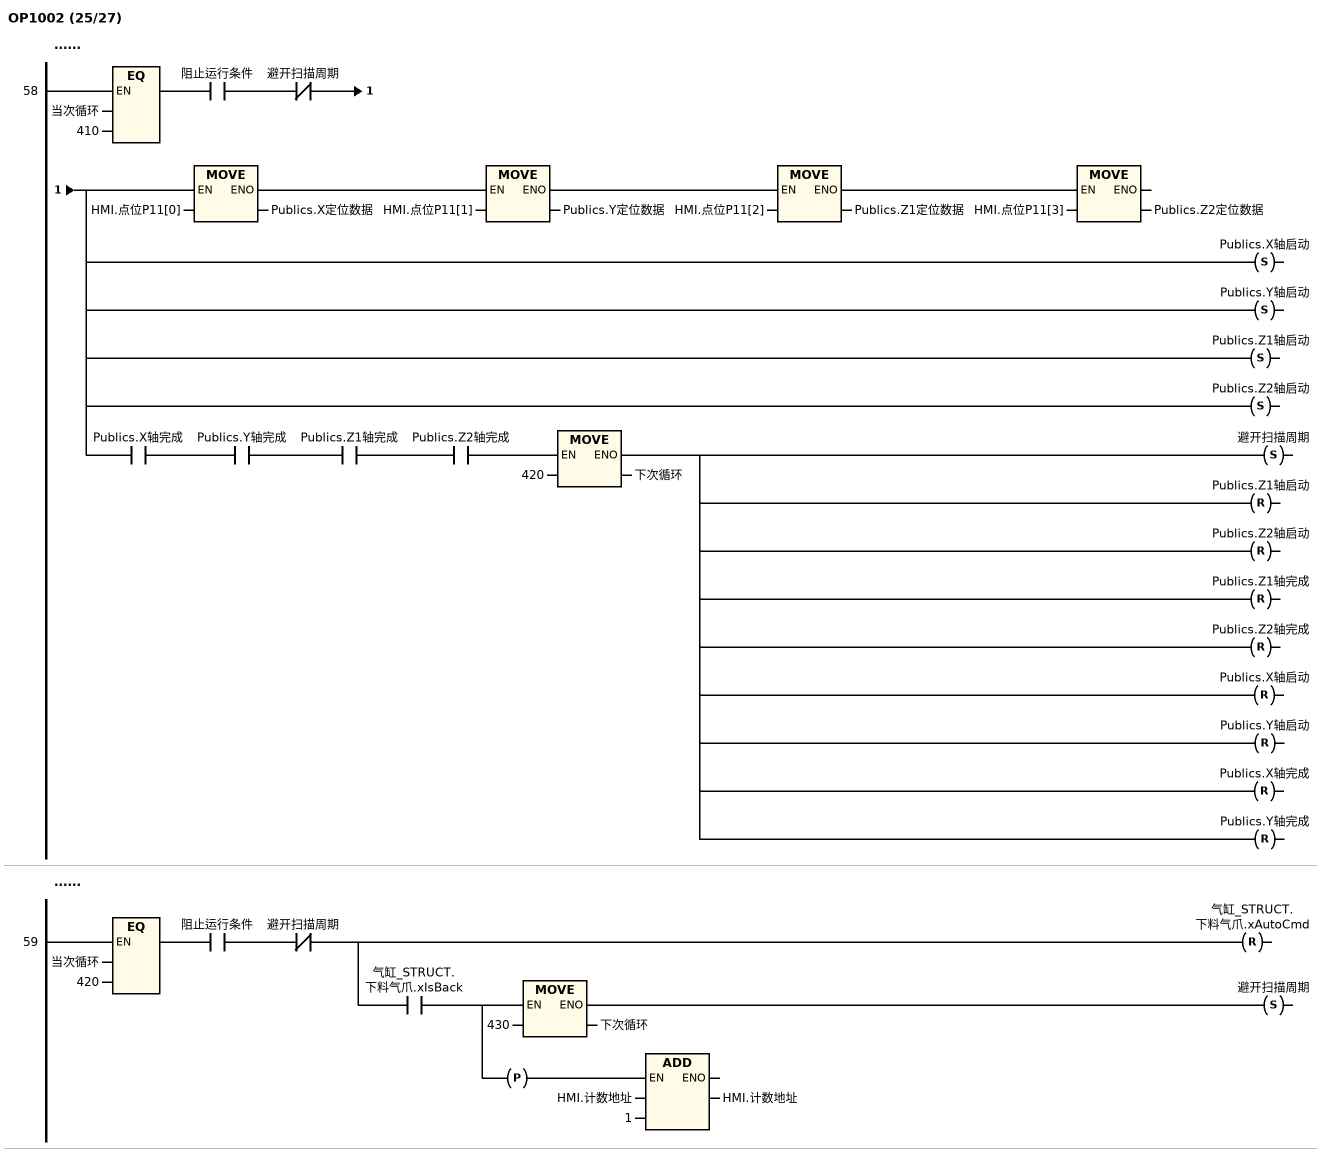
// NETWORK 58: ......
_w74 := 当次循环 = 410 AND 阻止运行条件 AND NOT 避开扫描周期;
IF _w74 THEN Publics.X定位数据 := HMI.点位P11[0]; END_IF
IF _w74 THEN Publics.Y定位数据 := HMI.点位P11[1]; END_IF
IF _w74 THEN Publics.Z1定位数据 := HMI.点位P11[2]; END_IF
IF _w74 THEN Publics.Z2定位数据 := HMI.点位P11[3]; END_IF
Publics.X轴启动 S= _w74;
Publics.Y轴启动 S= _w74;
Publics.Z1轴启动 S= _w74;
Publics.Z2轴启动 S= _w74;
IF _w74 AND Publics.X轴完成 AND Publics.Y轴完成 AND Publics.Z1轴完成 AND Publics.Z2轴完成 THEN 下次循环 := 420; END_IF
_w75 := _w74 AND Publics.X轴完成 AND Publics.Y轴完成 AND Publics.Z1轴完成 AND Publics.Z2轴完成;
避开扫描周期 S= _w75;
Publics.Z1轴启动 R= _w75;
Publics.Z2轴启动 R= _w75;
Publics.Z1轴完成 R= _w75;
Publics.Z2轴完成 R= _w75;
Publics.X轴启动 R= _w75;
Publics.Y轴启动 R= _w75;
Publics.X轴完成 R= _w75;
Publics.Y轴完成 R= _w75;

// NETWORK 59: ......
_w76 := 当次循环 = 420 AND 阻止运行条件 AND NOT 避开扫描周期;
气缸_STRUCT.下料气爪.xAutoCmd R= _w76;
_w77 := _w76 AND 气缸_STRUCT.下料气爪.xIsBack;
IF _w77 THEN 下次循环 := 430; END_IF
避开扫描周期 S= _w77;
_rt3(CLK := _w77);
IF _rt3.Q THEN HMI.计数地址 := HMI.计数地址 + 1; END_IF

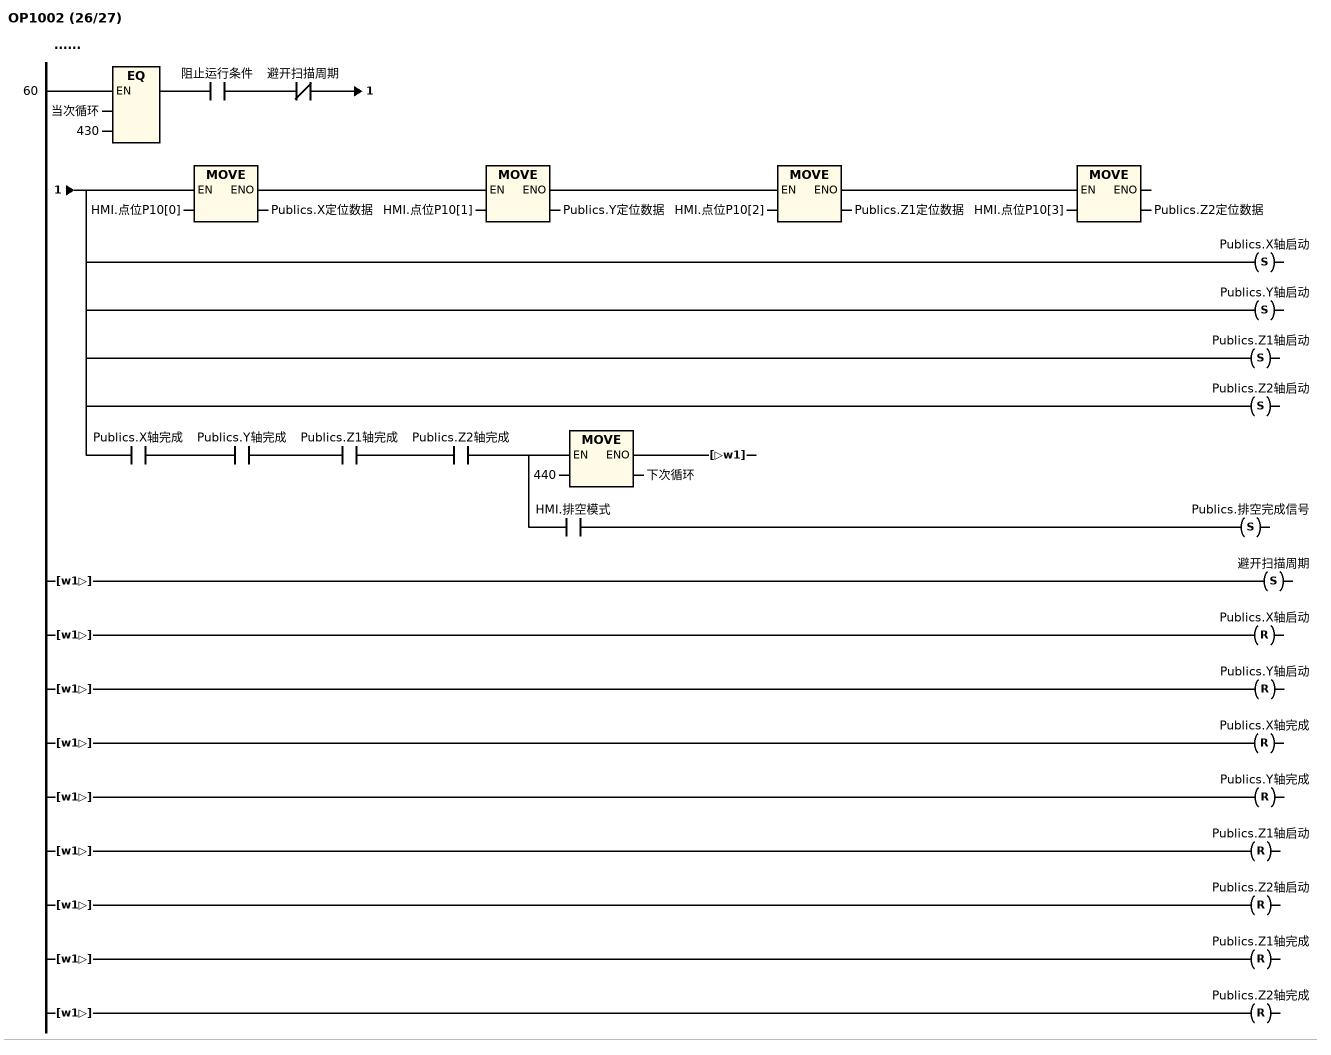
// NETWORK 60: ......
_w78 := 当次循环 = 430 AND 阻止运行条件 AND NOT 避开扫描周期;
IF _w78 THEN Publics.X定位数据 := HMI.点位P10[0]; END_IF
IF _w78 THEN Publics.Y定位数据 := HMI.点位P10[1]; END_IF
IF _w78 THEN Publics.Z1定位数据 := HMI.点位P10[2]; END_IF
IF _w78 THEN Publics.Z2定位数据 := HMI.点位P10[3]; END_IF
Publics.X轴启动 S= _w78;
Publics.Y轴启动 S= _w78;
Publics.Z1轴启动 S= _w78;
Publics.Z2轴启动 S= _w78;
_w79 := _w78 AND Publics.X轴完成 AND Publics.Y轴完成 AND Publics.Z1轴完成 AND Publics.Z2轴完成;
IF _w79 THEN 下次循环 := 440; END_IF
Publics.排空完成信号 S= _w79 AND HMI.排空模式;
避开扫描周期 S= _w79;
Publics.X轴启动 R= _w79;
Publics.Y轴启动 R= _w79;
Publics.X轴完成 R= _w79;
Publics.Y轴完成 R= _w79;
Publics.Z1轴启动 R= _w79;
Publics.Z2轴启动 R= _w79;
Publics.Z1轴完成 R= _w79;
Publics.Z2轴完成 R= _w79;

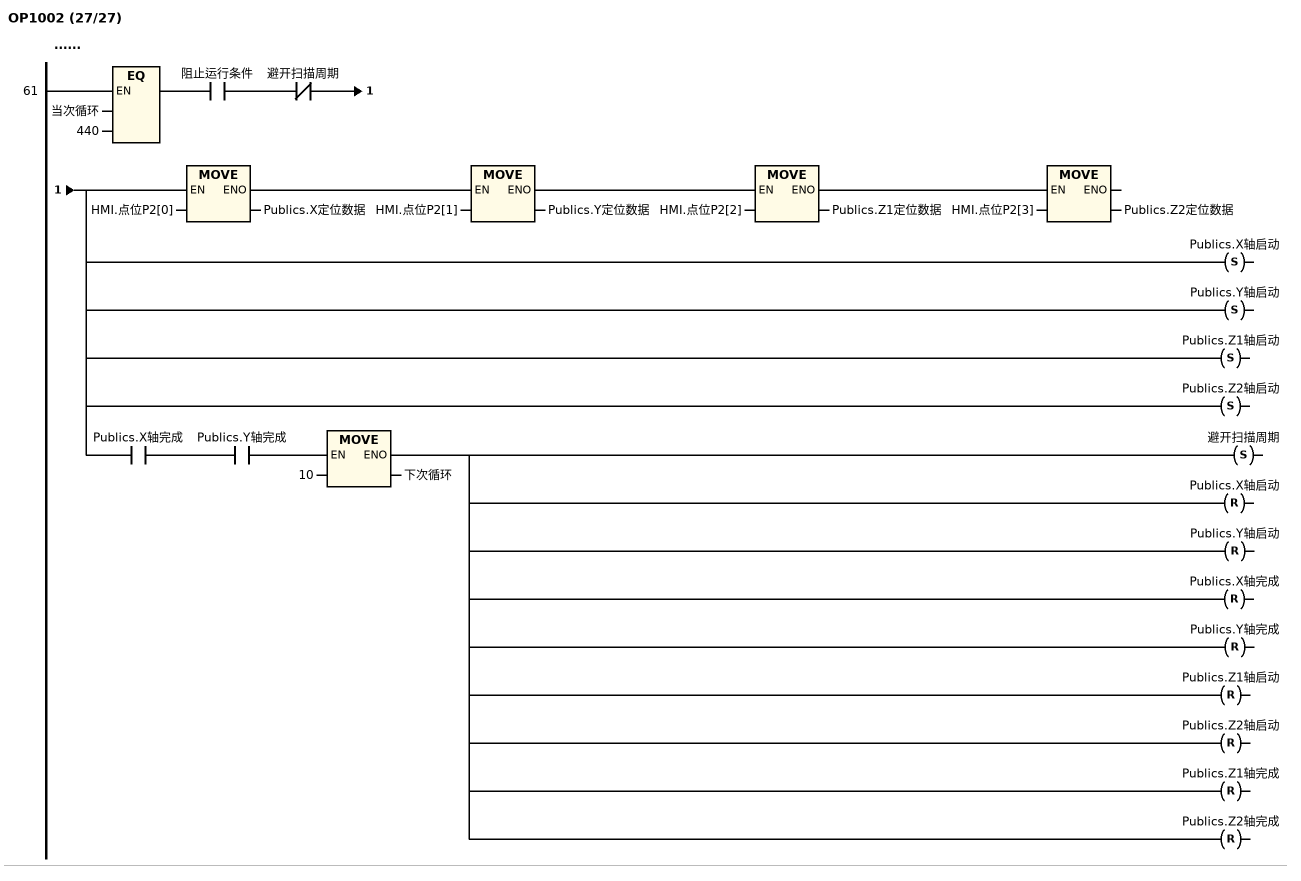
// NETWORK 61: ......
_w80 := 当次循环 = 440 AND 阻止运行条件 AND NOT 避开扫描周期;
IF _w80 THEN Publics.X定位数据 := HMI.点位P2[0]; END_IF
IF _w80 THEN Publics.Y定位数据 := HMI.点位P2[1]; END_IF
IF _w80 THEN Publics.Z1定位数据 := HMI.点位P2[2]; END_IF
IF _w80 THEN Publics.Z2定位数据 := HMI.点位P2[3]; END_IF
Publics.X轴启动 S= _w80;
Publics.Y轴启动 S= _w80;
Publics.Z1轴启动 S= _w80;
Publics.Z2轴启动 S= _w80;
IF _w80 AND Publics.X轴完成 AND Publics.Y轴完成 THEN 下次循环 := 10; END_IF
_w81 := _w80 AND Publics.X轴完成 AND Publics.Y轴完成;
避开扫描周期 S= _w81;
Publics.X轴启动 R= _w81;
Publics.Y轴启动 R= _w81;
Publics.X轴完成 R= _w81;
Publics.Y轴完成 R= _w81;
Publics.Z1轴启动 R= _w81;
Publics.Z2轴启动 R= _w81;
Publics.Z1轴完成 R= _w81;
Publics.Z2轴完成 R= _w81;

ACTION 辅助流程:
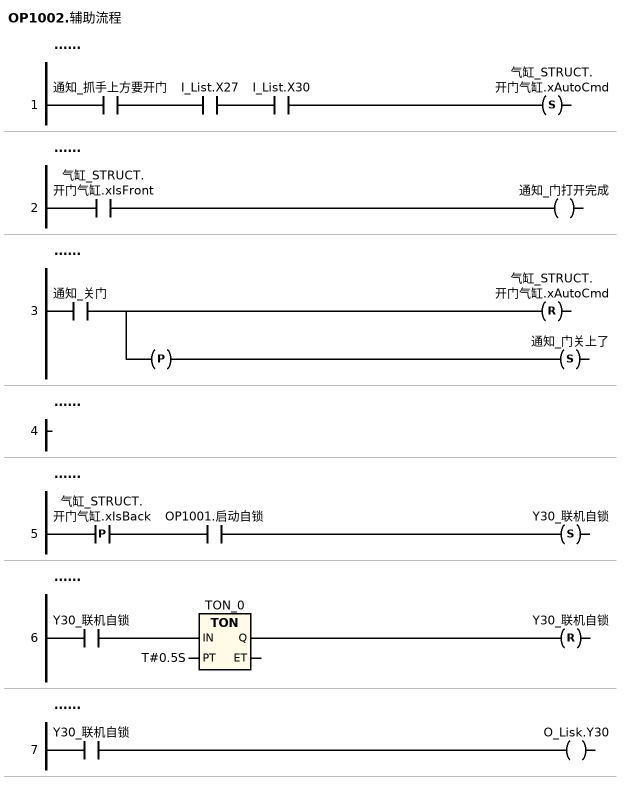
// NETWORK 1: ......
气缸_STRUCT.开门气缸.xAutoCmd S= 通知_抓手上方要开门 AND I_List.X27 AND I_List.X30;

// NETWORK 2: ......
通知_门打开完成 := 气缸_STRUCT.开门气缸.xIsFront;

// NETWORK 3: ......
气缸_STRUCT.开门气缸.xAutoCmd R= 通知_关门;
_rt4(CLK := 通知_关门);
通知_门关上了 S= _rt4.Q;

// NETWORK 4: ......

// NETWORK 5: ......
_rt5(CLK := 气缸_STRUCT.开门气缸.xIsBack);
Y30_联机自锁 S= _rt5.Q AND OP1001.启动自锁;

// NETWORK 6: ......
TON_0(IN := Y30_联机自锁, PT := T#0.5S); // TON
Y30_联机自锁 R= TON_0.Q;

// NETWORK 7: ......
O_Lisk.Y30 := Y30_联机自锁;
END_ACTION

END_PROGRAM

// Device/Application/气缸
PROGRAM 气缸
VAR
	FB_CylinderSingle_0: FB_CylinderSingle;
	上料推出气缸到位延时: word;
	上料推出气缸原位延时: word;
	FB_CylinderSingle_1: FB_CylinderSingle;
	上料推出气缸报警复位: BOOL;
	上料顶起气缸原位延时: WORD;
	上料顶起气缸到位位延时: WORD;
	FB_CylinderSingle_2: FB_CylinderSingle;
	FB_CylinderSingle_3: FB_CylinderSingle;
	FB_CylinderSingle_4: FB_CylinderSingle;
	FB_CylinderSingle_5: FB_CylinderSingle;
	FB_CylinderSingle_6: FB_CylinderSingle;
	A1: BOOL;
	A2: BOOL;
	A3: BOOL;
	A4: BOOL;
	A5: BOOL;
	A6: BOOL;
END_VAR
VAR // added by the converter: edge detectors and wires of the graphical bodies
    _rt1, _rt2, _rt3, _rt4, _rt5, _rt6, _rt7 : R_TRIG;
END_VAR

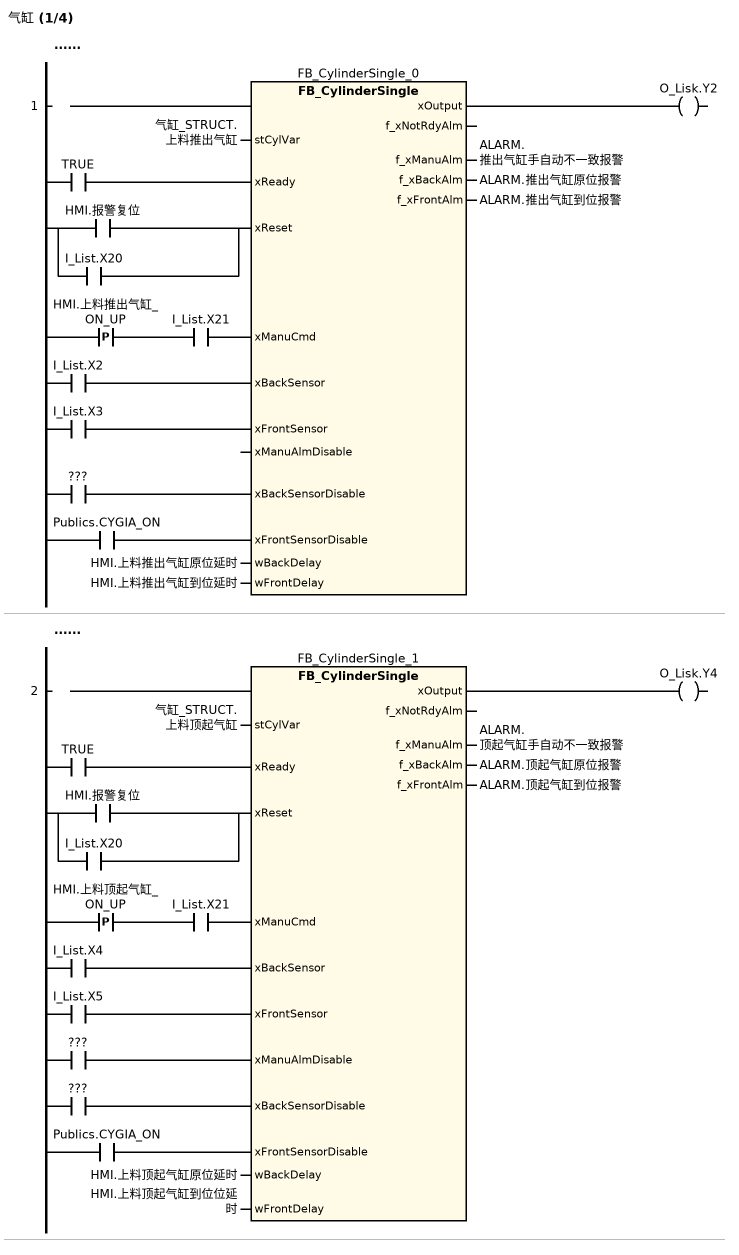
// NETWORK 1: ......
_rt1(CLK := HMI.上料推出气缸_ON_UP);
FB_CylinderSingle_0(
    stCylVar := 气缸_STRUCT.上料推出气缸,
    xReady := TRUE,
    xReset := HMI.报警复位 OR I_List.X20,
    xManuCmd := _rt1.Q AND I_List.X21,
    xBackSensor := I_List.X2,
    xFrontSensor := I_List.X3,
    xFrontSensorDisable := Publics.CYGIA_ON,
    wBackDelay := HMI.上料推出气缸原位延时,
    wFrontDelay := HMI.上料推出气缸到位延时,
    f_xManuAlm => ALARM.推出气缸手自动不一致报警,
    f_xBackAlm => ALARM.推出气缸原位报警,
    f_xFrontAlm => ALARM.推出气缸到位报警); // FB_CylinderSingle
O_Lisk.Y2 := FB_CylinderSingle_0.xOutput;

// NETWORK 2: ......
_rt2(CLK := HMI.上料顶起气缸_ON_UP);
FB_CylinderSingle_1(
    stCylVar := 气缸_STRUCT.上料顶起气缸,
    xReady := TRUE,
    xReset := HMI.报警复位 OR I_List.X20,
    xManuCmd := _rt2.Q AND I_List.X21,
    xBackSensor := I_List.X4,
    xFrontSensor := I_List.X5,
    xFrontSensorDisable := Publics.CYGIA_ON,
    wBackDelay := HMI.上料顶起气缸原位延时,
    wFrontDelay := HMI.上料顶起气缸到位位延时,
    f_xManuAlm => ALARM.顶起气缸手自动不一致报警,
    f_xBackAlm => ALARM.顶起气缸原位报警,
    f_xFrontAlm => ALARM.顶起气缸到位报警); // FB_CylinderSingle
O_Lisk.Y4 := FB_CylinderSingle_1.xOutput;

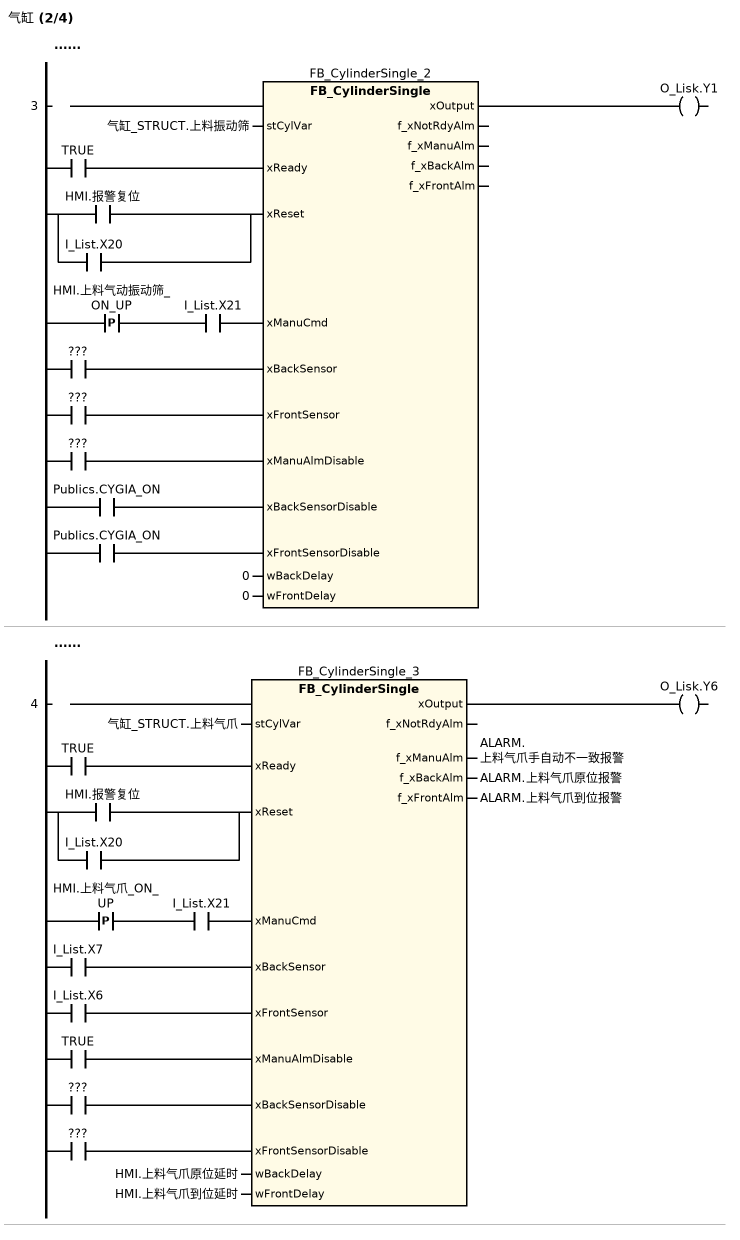
// NETWORK 3: ......
_rt3(CLK := HMI.上料气动振动筛_ON_UP);
FB_CylinderSingle_2(
    stCylVar := 气缸_STRUCT.上料振动筛,
    xReady := TRUE,
    xReset := HMI.报警复位 OR I_List.X20,
    xManuCmd := _rt3.Q AND I_List.X21,
    xBackSensorDisable := Publics.CYGIA_ON,
    xFrontSensorDisable := Publics.CYGIA_ON,
    wBackDelay := 0,
    wFrontDelay := 0); // FB_CylinderSingle
O_Lisk.Y1 := FB_CylinderSingle_2.xOutput;

// NETWORK 4: ......
_rt4(CLK := HMI.上料气爪_ON_UP);
FB_CylinderSingle_3(
    stCylVar := 气缸_STRUCT.上料气爪,
    xReady := TRUE,
    xReset := HMI.报警复位 OR I_List.X20,
    xManuCmd := _rt4.Q AND I_List.X21,
    xBackSensor := I_List.X7,
    xFrontSensor := I_List.X6,
    xManuAlmDisable := TRUE,
    wBackDelay := HMI.上料气爪原位延时,
    wFrontDelay := HMI.上料气爪到位延时,
    f_xManuAlm => ALARM.上料气爪手自动不一致报警,
    f_xBackAlm => ALARM.上料气爪原位报警,
    f_xFrontAlm => ALARM.上料气爪到位报警); // FB_CylinderSingle
O_Lisk.Y6 := FB_CylinderSingle_3.xOutput;

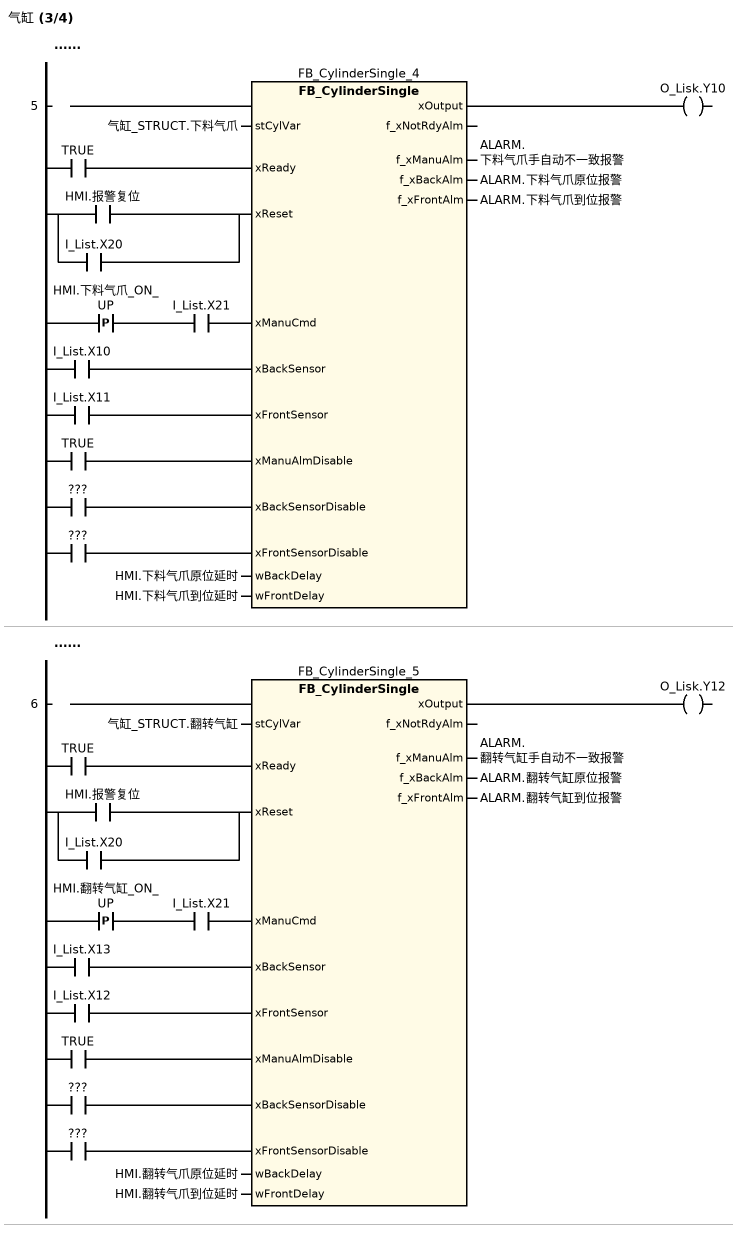
// NETWORK 5: ......
_rt5(CLK := HMI.下料气爪_ON_UP);
FB_CylinderSingle_4(
    stCylVar := 气缸_STRUCT.下料气爪,
    xReady := TRUE,
    xReset := HMI.报警复位 OR I_List.X20,
    xManuCmd := _rt5.Q AND I_List.X21,
    xBackSensor := I_List.X10,
    xFrontSensor := I_List.X11,
    xManuAlmDisable := TRUE,
    wBackDelay := HMI.下料气爪原位延时,
    wFrontDelay := HMI.下料气爪到位延时,
    f_xManuAlm => ALARM.下料气爪手自动不一致报警,
    f_xBackAlm => ALARM.下料气爪原位报警,
    f_xFrontAlm => ALARM.下料气爪到位报警); // FB_CylinderSingle
O_Lisk.Y10 := FB_CylinderSingle_4.xOutput;

// NETWORK 6: ......
_rt6(CLK := HMI.翻转气缸_ON_UP);
FB_CylinderSingle_5(
    stCylVar := 气缸_STRUCT.翻转气缸,
    xReady := TRUE,
    xReset := HMI.报警复位 OR I_List.X20,
    xManuCmd := _rt6.Q AND I_List.X21,
    xBackSensor := I_List.X13,
    xFrontSensor := I_List.X12,
    xManuAlmDisable := TRUE,
    wBackDelay := HMI.翻转气爪原位延时,
    wFrontDelay := HMI.翻转气爪到位延时,
    f_xManuAlm => ALARM.翻转气缸手自动不一致报警,
    f_xBackAlm => ALARM.翻转气缸原位报警,
    f_xFrontAlm => ALARM.翻转气缸到位报警); // FB_CylinderSingle
O_Lisk.Y12 := FB_CylinderSingle_5.xOutput;

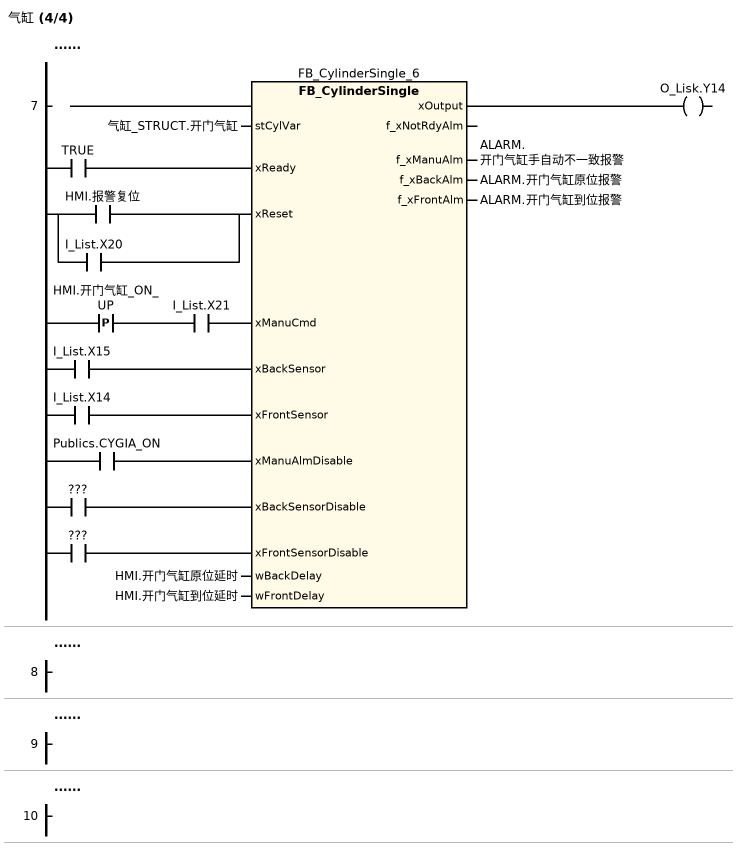
// NETWORK 7: ......
_rt7(CLK := HMI.开门气缸_ON_UP);
FB_CylinderSingle_6(
    stCylVar := 气缸_STRUCT.开门气缸,
    xReady := TRUE,
    xReset := HMI.报警复位 OR I_List.X20,
    xManuCmd := _rt7.Q AND I_List.X21,
    xBackSensor := I_List.X15,
    xFrontSensor := I_List.X14,
    xManuAlmDisable := Publics.CYGIA_ON,
    wBackDelay := HMI.开门气缸原位延时,
    wFrontDelay := HMI.开门气缸到位延时,
    f_xManuAlm => ALARM.开门气缸手自动不一致报警,
    f_xBackAlm => ALARM.开门气缸原位报警,
    f_xFrontAlm => ALARM.开门气缸到位报警); // FB_CylinderSingle
O_Lisk.Y14 := FB_CylinderSingle_6.xOutput;

// NETWORK 8: ......

// NETWORK 9: ......

// NETWORK 10: ......

END_PROGRAM

// Device/Application/FunctionBlock/FB_CylinderSingle
FUNCTION_BLOCK FB_CylinderSingle
VAR_IN_OUT
	stCylVar: CYLINDER_REF;
END_VAR
VAR_INPUT
	///安全条件
	xReady: BOOL;
	///报警复位
	xReset: BOOL;
	///手动控制,每on一次,则反转输出点状态
	xManuCmd: BOOL;
	///原位检测
	xBackSensor: BOOL;
	///到位检测
	xFrontSensor: BOOL;
	///手自动不一致报警无效
	xManuAlmDisable: BOOL;
	///原位检测无效
	xBackSensorDisable: BOOL;
	///到位检测无效
	xFrontSensorDisable: BOOL;
	///原位延时
	wBackDelay: WORD;
	///到位延时
	wFrontDelay: WORD;
END_VAR
VAR_OUTPUT
	xOutput: BOOL;
	///未满足安全条件报警
	f_xNotRdyAlm: BOOL;
	///手自动不一致报警	
	f_xManuAlm: BOOL;
	///未在原位报警
	f_xBackAlm: BOOL;
	///未到位报警
	f_xFrontAlm: BOOL;
END_VAR
VAR
	///获取自动控制的上升沿
	fbAutoRise: R_TRIG;
	///获取自动控制的下升沿
	fbAutoFall: F_TRIG;
	///获取手动控制的下升沿
	fbManuFall: F_TRIG;
	///获取复位信号的上升沿
	fbResetRise: R_TRIG;
	///原位状态延时,用于输出原位状态
	fbBackTon: TON;
	///到位状态延时,用于输出到位状态
	fbFrontTon: TON;
	///获取原位状态下降沿	
	fbBackFall: F_TRIG;
	///获取到位状态下降沿
	fbFrontFall: F_TRIG;
	///原位动作超时,用于输出未在原位位置报警
	fbBackWait: TON;
	///到位动作超时,用于输出未在到位位置报警
	fbFrontWait: TON;
END_VAR

   //初始化时复位输出点
   IF xReady AND stCylVar.xInit AND ( NOT f_xNotRdyAlm	) THEN
	    xOutput := FALSE;
	    f_xManuAlm  := FALSE;
	    stCylVar.xInit  := FALSE;
 
   END_IF


   //获取手动控制、自动控制的边沿信号
   fbManuFall(CLK:=xManuCmd , Q=> );
   fbAutoRise(CLK:=stCylvar.xAutoCmd , Q=> );
   fbAutoFall(CLK:=stCylvar.xAutoCmd , Q=> );
      
    //1,手动操作时，如果满足安全条件且未屏蔽了手自动不一致报警时，则输出点反转，  
    IF xReady AND (NOT xManuAlmDisable) AND fbManuFall.Q THEN
   	    xOutput  := NOT xOutput ;
		//手动操作生效时，判断输出点状态与自动命令是否一致，不一致时,置位手动操作执行中报警；一致时复位该报警。
	    //当因安全条件不满足导致自动命令未执行时，可通过手动操作控制其动作执行,此时手动操作并不引起手动操作执行中报警。
		 IF ( stCylvar.xAutoCmd ) XOR xOutput THEN
   	   	    f_xManuAlm  :=TRUE;
   	     ELSE 
   	   	    f_xManuAlm  :=FALSE;
   	     END_IF  	 	
     END_IF
	 
	//2,手动操作时，如果满足安全条件且屏蔽了手自动不一致报警时，则自动控制点反转、复位手自动不一致报警，  
    IF xReady AND  xManuAlmDisable AND fbManuFall.Q THEN
   	    stCylvar.xAutoCmd  := NOT stCylvar.xAutoCmd ;
		f_xManuAlm  :=FALSE;		  	 	
    END_IF
   
   
   
   //自动命令置位时，如果满足安全条件，则输出点置位
   IF xReady AND fbAutoRise.Q THEN
   	   xOutput  :=TRUE;
   END_IF
      
   //自动命令复位时，如满足安全条件，则输出点复位。
   IF xReady AND fbAutoFall.Q THEN
   	    xOutput  :=FALSE;		
   END_IF
   
   
   //原位状态输出
   fbBackTon(IN:= ( NOT xOutput) AND ( NOT xFrontSensor ) AND ( xBackSensor OR xBackSensorDisable ) , PT:= WORD_TO_TIME ( wBackDelay *10 ) , Q=> stCylvar.xIsBack, ET=> );
   
   
   //到位状态输出
   fbFrontTon(IN:= xOutput AND ( xFrontSensor OR xFrontSensorDisable ) AND ( NOT xBackSensor ) , PT:= WORD_TO_TIME ( wFrontDelay *10 ), Q=> stCylvar.xIsFront, ET=> );
      
	  
   //报警复位
   fbResetRise(CLK:= xReset, Q=> );
   IF fbResetRise.Q THEN
   	   f_xNotRdyAlm := FALSE;
	   f_xFrontAlm := FALSE;
	   f_xBackAlm := FALSE;
   
   END_IF
   
   
   //未满足安全条件报警
   //当手动操作或自动命令状态发生改变时，如果不能满足安全条件，则输出未满足安全条件报警
   IF ( fbManuFall.Q OR fbAutoRise.Q OR fbAutoFall.Q ) AND ( NOT xReady ) THEN
   	    f_xNotRdyAlm := TRUE; 
   END_IF
   
   
   //未在原位报警
   //自动命令变OFF后(上电后气缸处于自由状态时不判断)，延时5秒，如果原位标志未变为ON、且未发生手动操作和安全条件报警，则输出未到原位报警
   fbBackWait(IN:=  NOT stCylvar.xAutoCmd  , PT:= T#5S , Q=> , ET=> );
   fbBackFall(CLK:= stCylvar.xIsBack , Q=> );
   IF (( fbBackWait.Q AND (NOT stCylvar.xIsBack )) OR (( NOT stCylvar.xAutoCmd ) AND fbBackFall.Q )) AND  ( NOT f_xManuAlm ) AND  ( NOT f_xNotRdyAlm ) THEN
   	    f_xBackAlm := TRUE;
   END_IF
   
   
   //未到位报警
   //自动命令变ON后，延时5秒，如果到位标志未变为ON、且未发生手动操作和安全条件报警，则输出未到位报警
   fbFrontWait(IN:= stCylvar.xAutoCmd , PT:= T#5S , Q=> , ET=> );
   fbFrontFall(CLK:= stCylvar.xIsFront, Q=> );
   IF ( ( fbFrontWait.Q AND ( NOT stCylvar.xIsFront ) ) OR (stCylvar.xAutoCmd AND fbFrontFall.Q )) AND ( NOT f_xManuAlm ) AND ( NOT f_xNotRdyAlm ) THEN
   	    f_xFrontAlm := TRUE;   
   END_IF

END_FUNCTION_BLOCK

// Device/Application/其他手动
PROGRAM 其他手动
VAR
	手动皮带运转: BOOL;
	手动定位: BOOL;
END_VAR
VAR // added by the converter: edge detectors and wires of the graphical bodies
    _rt1 : R_TRIG;
    _w1, _w2, _w3, _w4, _w5, _w6, _w7, _w8, _w9, _w10, _w11, _w12, _w13, _w14 : BOOL;
END_VAR

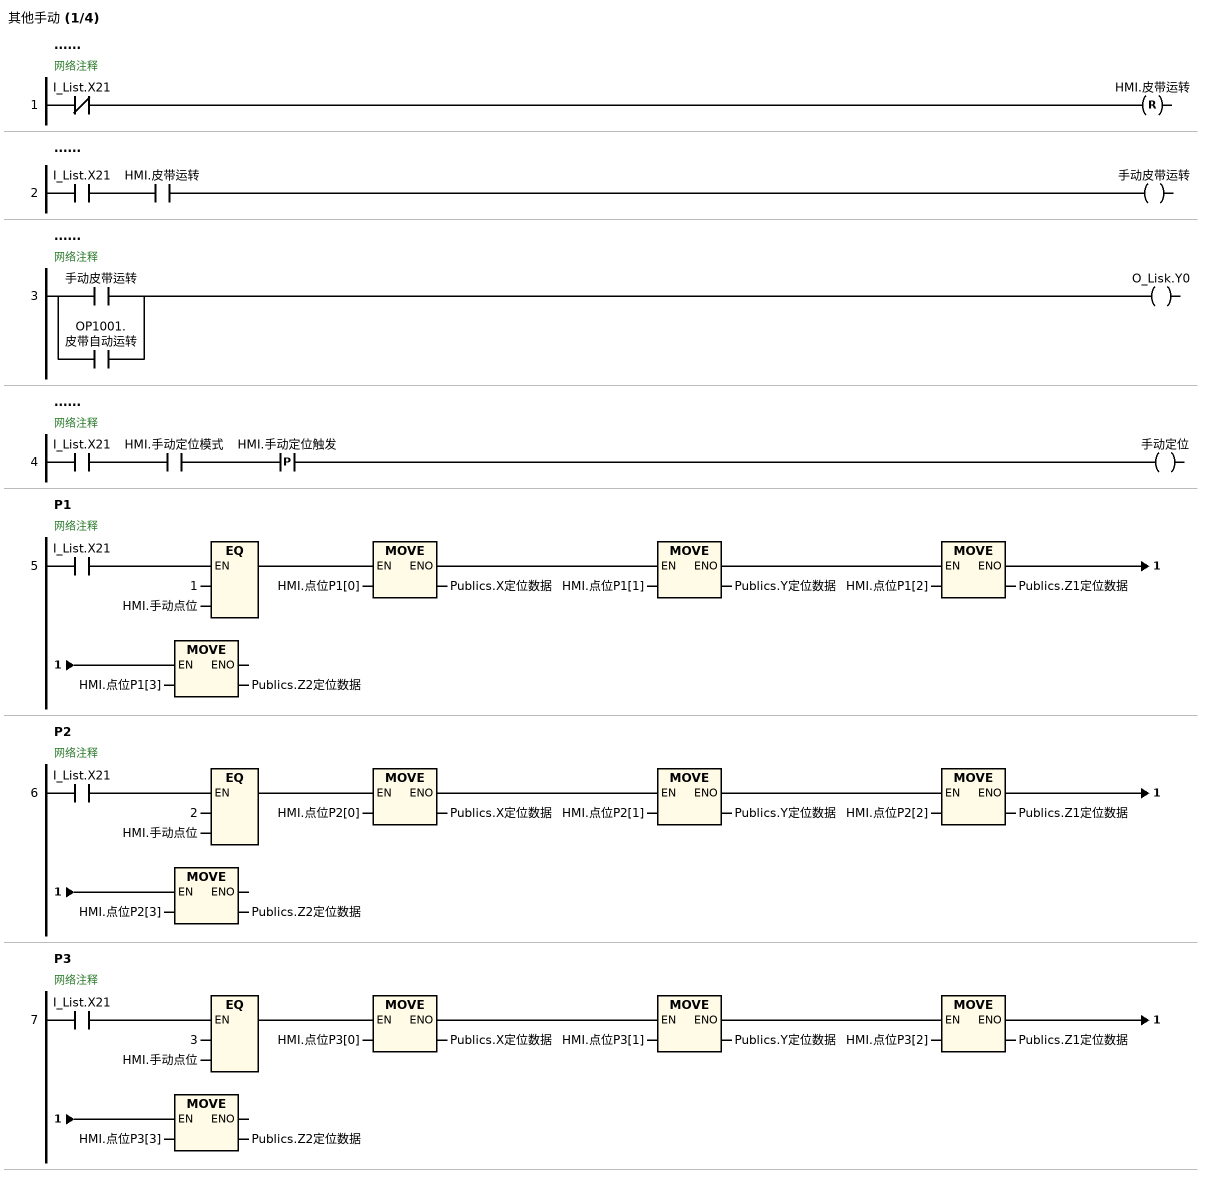
// NETWORK 1: ......
// 网络注释
HMI.皮带运转 R= NOT I_List.X21;

// NETWORK 2: ......
手动皮带运转 := I_List.X21 AND HMI.皮带运转;

// NETWORK 3: ......
// 网络注释
O_Lisk.Y0 := 手动皮带运转 OR OP1001.皮带自动运转;

// NETWORK 4: ......
// 网络注释
_rt1(CLK := HMI.手动定位触发);
手动定位 := I_List.X21 AND HMI.手动定位模式 AND _rt1.Q;

// NETWORK 5: P1
// 网络注释
_w1 := I_List.X21 AND 1 = HMI.手动点位;
IF _w1 THEN Publics.X定位数据 := HMI.点位P1[0]; END_IF
IF _w1 THEN Publics.Y定位数据 := HMI.点位P1[1]; END_IF
IF _w1 THEN Publics.Z1定位数据 := HMI.点位P1[2]; END_IF
IF _w1 THEN Publics.Z2定位数据 := HMI.点位P1[3]; END_IF

// NETWORK 6: P2
// 网络注释
_w2 := I_List.X21 AND 2 = HMI.手动点位;
IF _w2 THEN Publics.X定位数据 := HMI.点位P2[0]; END_IF
IF _w2 THEN Publics.Y定位数据 := HMI.点位P2[1]; END_IF
IF _w2 THEN Publics.Z1定位数据 := HMI.点位P2[2]; END_IF
IF _w2 THEN Publics.Z2定位数据 := HMI.点位P2[3]; END_IF

// NETWORK 7: P3
// 网络注释
_w3 := I_List.X21 AND 3 = HMI.手动点位;
IF _w3 THEN Publics.X定位数据 := HMI.点位P3[0]; END_IF
IF _w3 THEN Publics.Y定位数据 := HMI.点位P3[1]; END_IF
IF _w3 THEN Publics.Z1定位数据 := HMI.点位P3[2]; END_IF
IF _w3 THEN Publics.Z2定位数据 := HMI.点位P3[3]; END_IF

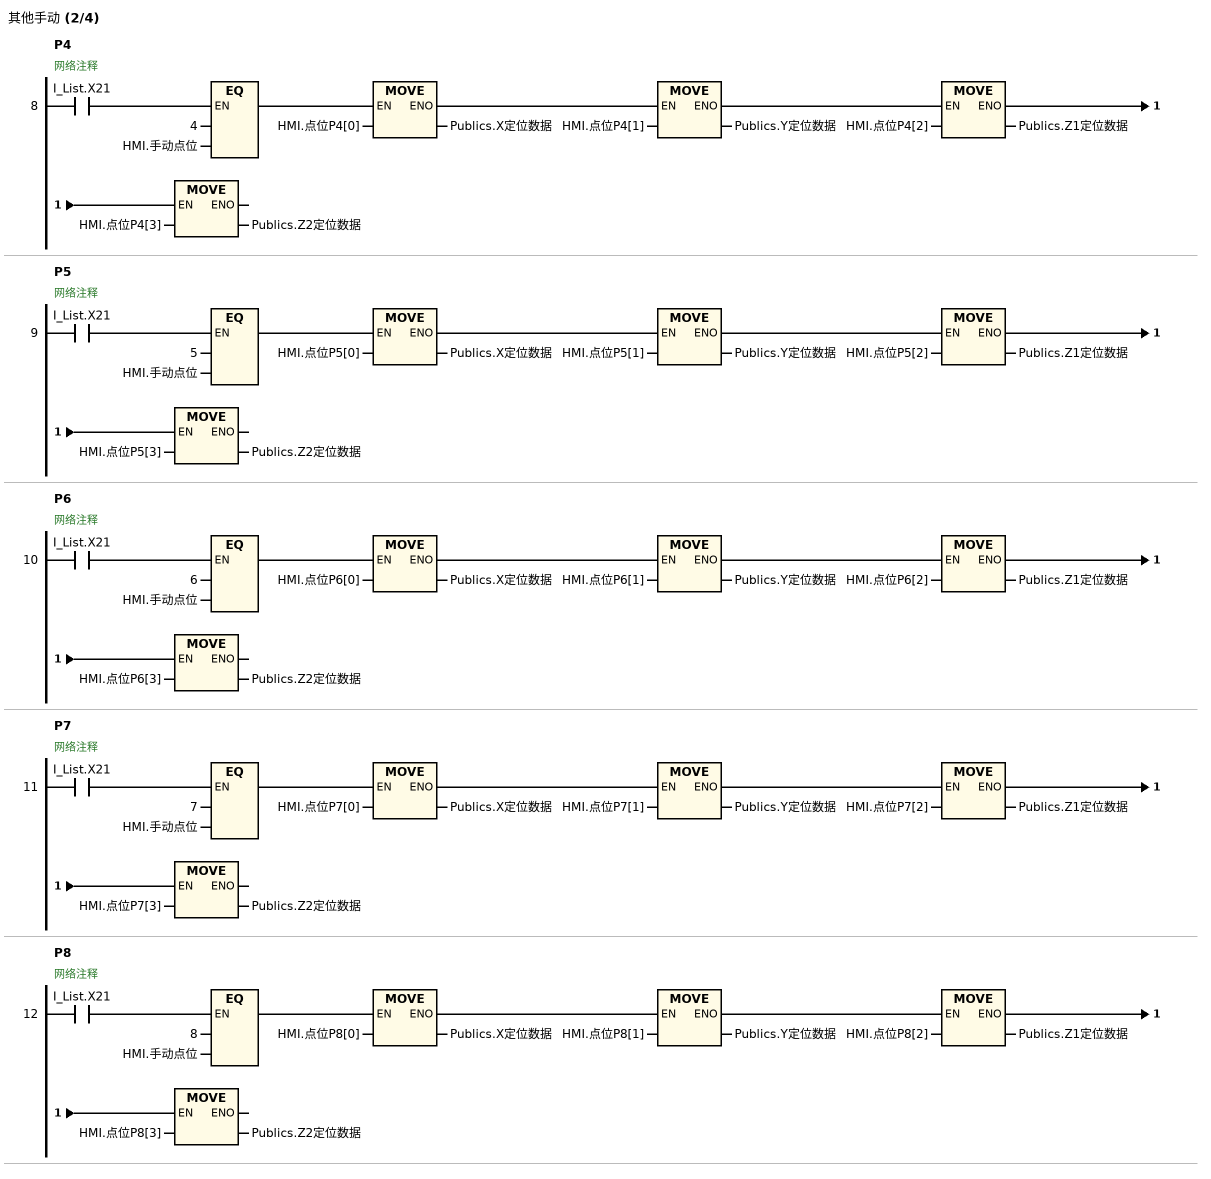
// NETWORK 8: P4
// 网络注释
_w4 := I_List.X21 AND 4 = HMI.手动点位;
IF _w4 THEN Publics.X定位数据 := HMI.点位P4[0]; END_IF
IF _w4 THEN Publics.Y定位数据 := HMI.点位P4[1]; END_IF
IF _w4 THEN Publics.Z1定位数据 := HMI.点位P4[2]; END_IF
IF _w4 THEN Publics.Z2定位数据 := HMI.点位P4[3]; END_IF

// NETWORK 9: P5
// 网络注释
_w5 := I_List.X21 AND 5 = HMI.手动点位;
IF _w5 THEN Publics.X定位数据 := HMI.点位P5[0]; END_IF
IF _w5 THEN Publics.Y定位数据 := HMI.点位P5[1]; END_IF
IF _w5 THEN Publics.Z1定位数据 := HMI.点位P5[2]; END_IF
IF _w5 THEN Publics.Z2定位数据 := HMI.点位P5[3]; END_IF

// NETWORK 10: P6
// 网络注释
_w6 := I_List.X21 AND 6 = HMI.手动点位;
IF _w6 THEN Publics.X定位数据 := HMI.点位P6[0]; END_IF
IF _w6 THEN Publics.Y定位数据 := HMI.点位P6[1]; END_IF
IF _w6 THEN Publics.Z1定位数据 := HMI.点位P6[2]; END_IF
IF _w6 THEN Publics.Z2定位数据 := HMI.点位P6[3]; END_IF

// NETWORK 11: P7
// 网络注释
_w7 := I_List.X21 AND 7 = HMI.手动点位;
IF _w7 THEN Publics.X定位数据 := HMI.点位P7[0]; END_IF
IF _w7 THEN Publics.Y定位数据 := HMI.点位P7[1]; END_IF
IF _w7 THEN Publics.Z1定位数据 := HMI.点位P7[2]; END_IF
IF _w7 THEN Publics.Z2定位数据 := HMI.点位P7[3]; END_IF

// NETWORK 12: P8
// 网络注释
_w8 := I_List.X21 AND 8 = HMI.手动点位;
IF _w8 THEN Publics.X定位数据 := HMI.点位P8[0]; END_IF
IF _w8 THEN Publics.Y定位数据 := HMI.点位P8[1]; END_IF
IF _w8 THEN Publics.Z1定位数据 := HMI.点位P8[2]; END_IF
IF _w8 THEN Publics.Z2定位数据 := HMI.点位P8[3]; END_IF

